// ---- 01_Equipement_Library/Sensors/TOR/FB_TOR_Spd.TcPOU
FUNCTION_BLOCK FB_TOR_Spd EXTENDS FB_TOR_Base
//////////////////
//  Surge Protection Device
//////////////////
VAR_INPUT PERSISTENT
	// Parameters of the Object (instance/model specific) 
	ParamTempoEs :TIME:=T#5S;(*  (s)Tempo before raising an alarm*)
END_VAR

VAR_OUTPUT
	//Child objects
	
END_VAR

VAR_INPUT
	// I/O Inputs 		                                     				
		
			MesDataExd			: TOR_Standard ;  

END_VAR

VAR
	//M_ALARMMANAGEMENT VARIABLES//
		FB_PermAlarm				: SR ;					// (NA) FB to maintain Fire Alarm even if sensor stop detection (burn) .
		TON_ES						: TON ; 
 
	//M_STATEMANAGER VARIABLES//

		
END_VAR

METHOD M_AlarmManagement
//////////////////
// Manages Smoke detector alarms and warnings
/////////////////

VAR 
	// Method local variables (reinitialized at each cycle) 
	FB_AlarmCodeManager			: FB_AlarmCodeManager ; 

END_VAR
// Detection Variables
TON_ES(IN:= MesDataExd.MesData.MesAlarmState , PT:= ParamTempoEs ) ; 
FB_PermAlarm(SET1 := TON_ES.Q  , Reset := CmdClearFault_G OR IN_CmdReset_L ); // SR FB for keep fire if burn .

// ALARM CODE //
	FB_AlarmCodeManager(
		bAlarm1			:= FB_PermAlarm.Q1 ,  														// Surge protection triggered	
		bAlarm2			:= SEL(ParamNbSensors<>1,FALSE, IN_MesState1_IO <> IN_MesState2_IO), 		// UNcoherent measure
		bAlarm3			:=FALSE, 																	// 
		bAlarm4			:=FALSE, 																	// 
		bAlarm5			:=FALSE, 																	//	
		bAlarm6			:=FALSE,                                                                    //
		bAlarm7			:=FALSE,                                                                    //
		bAlarm8			:=FALSE,                                                                    //
		bAlarm9			:=FALSE,                                                                    //
		bAlarm10		:=FALSE,                                                                    //
		bAlarm11		:=FALSE,                                                                    //
		bAlarm12		:=FALSE,                                                                    //
		bAlarm13		:=FALSE,                                                                    //
		bAlarm14		:=FALSE,                                                                    //
		bAlarm15		:=FALSE,                                                                    //
		wAlarmCode		=>MesDataExd.MesData.MesAlarmCode );
		
// WARNING CODE //
	FB_AlarmCodeManager(
		bAlarm1			:= IN_MesState1_IO OR  IN_MesState2_IO,	  									// At least one detector is ON 
		bAlarm2			:=FALSE, 																	// 
		bAlarm3			:=FALSE, 																	// 
		bAlarm4			:=FALSE, 																	// 
		bAlarm5			:=FALSE, 																	//
		bAlarm6			:=FALSE,        															//
		bAlarm7			:=FALSE,        															//
		bAlarm8			:=FALSE,        															//
		bAlarm9			:=FALSE,        															//
		bAlarm10		:=FALSE,        															//
		bAlarm11		:=FALSE,        															//
		bAlarm12		:=FALSE,        															//
		bAlarm13		:=FALSE,        															//
		bAlarm14		:=FALSE,        															//
		bAlarm15		:=FALSE,        															//
		wAlarmCode			=>MesDataExd.MesData.MesWarningCode);
		
// EVENT CODE //
	FB_AlarmCodeManager(
		bAlarm1			:= IN_MesState1_IO, 															// First sensor is ON
		bAlarm2			:= IN_MesState2_IO, 															// Second sensor is ON
		bAlarm3			:= FALSE, 																		// 
		bAlarm4			:= FALSE, 																		// 
		bAlarm5			:= FALSE, 																		//			
		bAlarm6			:= FALSE,                           											//
		bAlarm7			:= FALSE,                           											//
		bAlarm8			:= FALSE,                           											//
		bAlarm9			:= FALSE,                           											//
		bAlarm10		:= FALSE,                           											//
		bAlarm11		:= FALSE,                           											//
		bAlarm12		:= FALSE,                           											//
		bAlarm13		:= FALSE,                           											//
		bAlarm14		:= FALSE,                           											//
		bAlarm15		:= FALSE,                           											//
		wAlarmCode		=>MesDataExd.MesData.MesEventCode);
END_METHOD

METHOD M_Execute
//////////////////
//  Method Calls 
/////////////////

VAR 
	// Method local variables (reinitialized at each cycle) 

END_VAR

	
	IF ParamNbSensors = 9 THEN // Use of contactor bi-stable No and NC
		IN_MesState2_IO := NOT IN_MesState2_IO;
	END_IF
SUPER^.M_Execute() ;
END_METHOD

METHOD M_Init
VAR_INPUT
END_VAR
//A1_SPD_Aux.ParamAtleastOne := TRUE ; 
//A1_SPD_Aux.ParamNbSensors := 1 ; 
//A1_SPD_Aux.ParamCableCutSecurity := TRUE ;
END_METHOD

METHOD M_StateManager
//////////////////
// Detect when fire occurs
/////////////////

VAR 
	// Method local variables (reinitialized at each cycle)
 	MesStateInterm1 : BOOL;
	MesStateInterm2 : BOOL;
END_VAR

IF ParamCableCutSecurity THEN
	MesStateInterm1 := NOT IN_MesState1_IO ; 
	MesStateInterm2 := NOT IN_MesState2_IO ; 
ELSE 
	MesStateInterm1 := IN_MesState1_IO;
	MesStateInterm2 := IN_MesState2_IO;
END_IF

IF ParamNbSensors = 1 THEN 
	MesStateInterm2 := MesStateInterm1 ;
END_IF

IF ParamAtleastOne THEN 
MesDataExd.MesData.MesAlarmState := MesStateInterm1 OR MesStateInterm2 ; 
ELSE
MesDataExd.MesData.MesAlarmState := MesStateInterm1 AND MesStateInterm2 ; 
END_IF

R_TRIGAlarm(CLK:= MesDataExd.MesData.MesAlarmState ) ; 
IF R_TRIGAlarm.Q THEN
	MesCountAlarm :=  MIN(MesCountAlarm + 1 ,4294967295 ) ; 
ELSIF IN_ResetCounter THEN 
	MesCountAlarm := 0 ; 
END_IF

MesDataExd.MesData.MesCountAlarm	:= MesCountAlarm ;
END_METHOD

END_FUNCTION_BLOCK

// ---- 01_Equipement_Library/Sensors/TOR/FB_TOR_VP.TcPOU
FUNCTION_BLOCK FB_TOR_VP EXTENDS FB_TOR_Base
//////////////////
//  Voltage Presence
//////////////////

VAR_INPUT PERSISTENT
	// Parameters of the Object (instance/model specific) 
		
		
END_VAR

VAR_OUTPUT
	//Child objects
	
END_VAR

VAR_INPUT
	// I/O Inputs 		                                     				
		MesDataExd			: TOR_Standard ;  

END_VAR

VAR
	//M_ALARMMANAGEMENT VARIABLES//
		

	
END_VAR

METHOD M_AlarmManagement
//////////////////
// Manages Door sensor alarms and warnings
/////////////////

VAR 
	// Method local variables (reinitialized at each cycle) 
	FB_AlarmCodeManager : FB_AlarmCodeManager ; 


END_VAR

// ALARM CODE //
	FB_AlarmCodeManager(
 		bAlarm1			:= FALSE,    					// 
		bAlarm2			:= FALSE, 						// 
		bAlarm3			:= FALSE, 						// 
		bAlarm4			:= FALSE, 						// 
		bAlarm5			:= FALSE,       				//
		bAlarm6			:= FALSE,       				//
		bAlarm7			:= FALSE,       				//
		bAlarm8			:= FALSE,       				//
		bAlarm9			:= FALSE,       				//
		bAlarm10		:= FALSE,       				//
		bAlarm11		:= FALSE,       				//
		bAlarm12		:= FALSE,         				//
		bAlarm13		:= FALSE,         				//
		bAlarm14		:= FALSE,         				//
		bAlarm15		:= FALSE,         				//
		wAlarmCode		=>MesDataExd.MesData.MesAlarmCode);

// WARNING CODE //
	FB_AlarmCodeManager(
		bAlarm1			:= FALSE,    			// 
		bAlarm2			:= FALSE, 				//  
		bAlarm3			:= FALSE, 				//  
		bAlarm4			:= FALSE, 				//  
		bAlarm5			:= FALSE,               //
		bAlarm6			:= FALSE,               //
		bAlarm7			:= FALSE,               //
		bAlarm8			:= FALSE,               //
		bAlarm9			:= FALSE,               //
		bAlarm10		:= FALSE,               //
		bAlarm11		:= FALSE,               //
		bAlarm12		:= FALSE,               //
		bAlarm13		:= FALSE,               //
		bAlarm14		:= FALSE,               //
		bAlarm15		:= FALSE,               //
		wAlarmCode		=>MesDataExd.MesData.MesWarningCode);

// EVENT CODE //
	FB_AlarmCodeManager(
		bAlarm1			:= MesDataExd.MesData.MesAlarmState, 			//  Voltage not present anymore
		bAlarm2			:= FALSE, 							// 
		bAlarm3			:= FALSE, 							//  
		bAlarm4			:= FALSE, 							// 
		bAlarm5			:= FALSE,                           //
		bAlarm6			:= FALSE,                           //
		bAlarm7			:= FALSE,                           //
		bAlarm8			:= FALSE,                           //
		bAlarm9			:= FALSE,                           //
		bAlarm10		:= FALSE,                           //
		bAlarm11		:= FALSE,                           //
		bAlarm12		:= FALSE,                           //
		bAlarm13		:= FALSE,                           //
		bAlarm14		:= FALSE,                           //
		bAlarm15		:= FALSE,                           //
		wAlarmCode		=>MesDataExd.MesData.MesEventCode);
END_METHOD

METHOD M_StateManager
//////////////////
// Detect when fire occurs
/////////////////

VAR 
	// Method local variables (reinitialized at each cycle)
 	MesStateInterm1 : BOOL;
	MesStateInterm2 : BOOL;
END_VAR

IF ParamCableCutSecurity THEN
	MesStateInterm1 := NOT IN_MesState1_IO ; 
	MesStateInterm2 := NOT IN_MesState2_IO ; 
ELSE 
	MesStateInterm1 := IN_MesState1_IO;
	MesStateInterm2 := IN_MesState2_IO;
END_IF

IF ParamNbSensors = 1 THEN 
	MesStateInterm2 := MesStateInterm1 ;
END_IF

IF ParamAtleastOne THEN 
MesDataExd.MesData.MesAlarmState := MesStateInterm1 OR MesStateInterm2 ; 
ELSE
MesDataExd.MesData.MesAlarmState := MesStateInterm1 AND MesStateInterm2 ; 
END_IF

R_TRIGAlarm(CLK:= MesDataExd.MesData.MesAlarmState ) ; 
IF R_TRIGAlarm.Q THEN
	MesCountAlarm :=  MIN(MesCountAlarm + 1 ,4294967295 ) ; 
ELSIF IN_ResetCounter THEN 
	MesCountAlarm := 0 ; 
END_IF

MesDataExd.MesData.MesCountAlarm	:= MesCountAlarm ;
END_METHOD

END_FUNCTION_BLOCK

// ---- 01_Equipement_Library/Sensors/TOR/FB_TOR_DS.TcPOU
FUNCTION_BLOCK FB_TOR_DS EXTENDS FB_TOR_Base
//////////////////
//  Door sensor system . State = True >> Door Closed .
//////////////////

VAR_INPUT PERSISTENT
	// Parameters of the Object (instance/model specific) 
		ParamTempoDoorAlarm			: TIME := T#10S ;	(* (s) Tempo for Door sensor alarm *)
		
END_VAR

VAR_OUTPUT
	//Child objects
	
END_VAR

VAR_INPUT
	// I/O Inputs 		                                     				
	MesDataExd			: TOR_Standard ;  
		
END_VAR

VAR
	//M_ALARMMANAGEMENT VARIABLES//
		TON_Ouverture				: TON;				//(NA) Tempo to detect door opened for too long time . 



END_VAR

METHOD M_AlarmManagement
//////////////////
// Manages Door sensor alarms and warnings
/////////////////

VAR 
	// Method local variables (reinitialized at each cycle) 
	FB_AlarmCodeManager : FB_AlarmCodeManager ; 


END_VAR
// Detection Variables
TON_Ouverture(IN:= MesDataExd.MesData.MesAlarmState,PT:=ParamTempoDoorAlarm);

// ALARM CODE //
	FB_AlarmCodeManager(
 		bAlarm1			:= FALSE,    	// 
		bAlarm2			:= FALSE, 		// 
		bAlarm3			:= FALSE, 		// 
		bAlarm4			:= FALSE, 		// 
		bAlarm5			:= FALSE,       //
		bAlarm6			:= FALSE,       //
		bAlarm7			:= FALSE,       //
		bAlarm8			:= FALSE,       //
		bAlarm9			:= FALSE,       //
		bAlarm10		:= FALSE,       //
		bAlarm11		:= FALSE,       //
		bAlarm12		:= FALSE,       //
		bAlarm13		:= FALSE,       //
		bAlarm14		:= FALSE,       //
		bAlarm15		:= FALSE,       //
		wAlarmCode		=>MesDataExd.MesData.MesAlarmCode);

// WARNING CODE //
	FB_AlarmCodeManager(
		bAlarm1			:= TON_Ouverture.Q,    	// The door is opened for more than 15 seconds
		bAlarm2			:= FALSE, 				// 
		bAlarm3			:= FALSE, 				// 
		bAlarm4			:= FALSE, 				// 
		bAlarm5			:= FALSE, 				//
		bAlarm6			:= FALSE,               //
		bAlarm7			:= FALSE,               //
		bAlarm8			:= FALSE,               //
		bAlarm9			:= FALSE,               //
		bAlarm10		:= FALSE,               //
		bAlarm11		:= FALSE,               //
		bAlarm12		:= FALSE,               //
		bAlarm13		:= FALSE,               //
		bAlarm14		:= FALSE,               //
		bAlarm15		:= FALSE,               //
		wAlarmCode		=>MesDataExd.MesData.MesWarningCode);

// EVENT CODE //
	FB_AlarmCodeManager(
		bAlarm1			:= MesDataExd.MesData.MesAlarmState, 		// Door is Opened
		bAlarm2			:= FALSE, 						// 
		bAlarm3			:= FALSE, 						// 
		bAlarm4			:= FALSE, 						// 
		bAlarm5			:= FALSE, 						//
		bAlarm6			:= FALSE, 						//
		bAlarm7			:= FALSE, 						//
		bAlarm8			:= FALSE, 						//
		bAlarm9			:= FALSE, 						//
		bAlarm10		:= FALSE, 						//
		bAlarm11		:= FALSE, 						//
		bAlarm12		:= FALSE, 						//
		bAlarm13		:= FALSE, 						//
		bAlarm14		:= FALSE, 						//
		bAlarm15		:= FALSE, 						//
		wAlarmCode		=>MesDataExd.MesData.MesEventCode);
END_METHOD

METHOD M_Execute
//////////////////
//  Method Calls 
/////////////////

VAR 
	// Method local variables (reinitialized at each cycle) 
	
END_VAR


SUPER^.M_Execute() ;
END_METHOD

METHOD M_StateManager
//////////////////
// Detect when fire occurs
/////////////////

VAR 
	// Method local variables (reinitialized at each cycle)
 	MesStateInterm1 : BOOL;
	MesStateInterm2 : BOOL;
END_VAR

IF ParamCableCutSecurity THEN
	MesStateInterm1 := NOT IN_MesState1_IO ; 
	MesStateInterm2 := NOT IN_MesState2_IO ; 
ELSE 
	MesStateInterm1 := IN_MesState1_IO;
	MesStateInterm2 := IN_MesState2_IO;
END_IF

IF ParamNbSensors = 1 THEN 
	MesStateInterm2 := MesStateInterm1 ;
END_IF

IF ParamAtleastOne THEN 
MesDataExd.MesData.MesAlarmState := MesStateInterm1 OR MesStateInterm2 ; 
ELSE
MesDataExd.MesData.MesAlarmState := MesStateInterm1 AND MesStateInterm2 ; 
END_IF

R_TRIGAlarm(CLK:= MesDataExd.MesData.MesAlarmState ) ; 
IF R_TRIGAlarm.Q THEN
	MesCountAlarm :=  MIN(MesCountAlarm + 1 ,4294967295 ) ; 
ELSIF IN_ResetCounter THEN 
	MesCountAlarm := 0 ; 
END_IF

MesDataExd.MesData.MesCountAlarm	:= MesCountAlarm ;
END_METHOD

END_FUNCTION_BLOCK

// ---- 01_Equipement_Library/Sensors/TOR/FB_TOR_Rain.TcPOU
FUNCTION_BLOCK FB_TOR_Rain EXTENDS FB_TOR_Base
//////////////////
//  Rain sensor system.
//////////////////

VAR_INPUT PERSISTENT
	// Parameters of the Object (instance/model specific) 
	ParamRainPerPulse				: REAL := 10 ; (* (mm) Number of mm of rain per pulse		*)
END_VAR

VAR_OUTPUT
	//Child objects
	
END_VAR

VAR_INPUT
	// I/O Inputs 		                                     				
    ParamVarHrWarning   			: REAL :=8 ;  // (mm) Max of raining before warning mm of rain for last hour --> Mean it is raining a lot  Defaut value 8       
    ParamVarDayWarning  			: REAL :=48;  // (mm )max of raining before warning mm of rain for last day  --> Mean it rained a lot during 1 day defaut value 48
	ParamVarMinAlarm				: REAL :=-5;  // (%)  Config : Minimal allowed Site Hygrometry 



	MesDataExd			: TOR_Rain;
END_VAR

VAR


	//M_ALARMMANAGEMENT VARIABLES//
		WarningDay					: BOOL;
		WarningHr					: BOOL;
		WarningValue				: BOOL;
	
	
	//M_Execute
		FB_AverageHr				: FB_Average; 	
	    FB_AverageDay               : FB_Average;
	    FB_AverageMonth             : FB_Average;
		CTUHr						: CTU;
		CTUDay						: CTU;
		CTUMonth					: CTU;
		Hour 						: INT;
		PluvioHr_Avg		        : REAL ; 
		PluvioDay_Avg		        : REAL ; 
		PluvioMonth_Avg		        : REAL ;     
		PluvioHr_Max		        : REAL;
		PluvioDay_Max		        : REAL ; 
		PluvioMonth_Max		        : REAL ; 
        PluvioHr					: REAL ; 
		PluvioDay					: REAL ; 
		PluvioMonth					: REAL ; 

	
	
END_VAR

METHOD M_AlarmManagement
//////////////////
// Manages Door sensor alarms and warnings
/////////////////

VAR 
	// Method local variables (reinitialized at each cycle) 
	FB_AlarmCodeManager : FB_AlarmCodeManager ; 
END_VAR
	WarningDay	:= PluvioDay >= ParamVarDayWarning;
	WarningHr	:= PluvioHr >= ParamVarHrWarning;
	WarningValue:= PluvioDay <= ParamVarMinAlarm OR PluvioHr <= ParamVarMinAlarm;

// ALARM CODE //
	FB_AlarmCodeManager(
 		bAlarm1			:= FALSE,    								// 
		bAlarm2			:= FALSE, 									// 
		bAlarm3			:= FALSE, 									// 
		bAlarm4			:= FALSE, 									// 
		bAlarm5			:= FALSE,     								//
		bAlarm6			:= FALSE,  									//
		bAlarm7			:= FALSE,  									//
		bAlarm8			:= FALSE,  									//
		bAlarm9			:= FALSE,    								// 
		bAlarm10		:= FALSE, 									// 
		bAlarm11		:= FALSE, 									// 
		bAlarm12		:= FALSE, 									// 
		bAlarm13		:= FALSE,									// 
		bAlarm14		:= FALSE,									// 
		bAlarm15		:= FALSE,									// 
		wAlarmCode		=>MesDataExd.MesData.MesAlarmCode);

// WARNING CODE //
	FB_AlarmCodeManager(
		bAlarm1			:= WarningHr,   							// Raining too hard 
		bAlarm2			:= WarningDay, 								// Raining a lot during one day
		bAlarm3			:= WarningValue, 							// Raining value not coherent
		bAlarm4			:= FALSE, 									// 
		bAlarm5			:= FALSE,    								// 
		bAlarm6			:= FALSE, 									// 
		bAlarm7			:= FALSE, 									// 
		bAlarm8			:= FALSE, 									// 
		bAlarm9			:= FALSE,    								// 
		bAlarm10		:= FALSE, 									// 
		bAlarm11		:= FALSE, 									// 
		bAlarm12		:= FALSE, 									// 
		bAlarm13		:= FALSE,									// 
		bAlarm14		:= FALSE,									// 
		bAlarm15		:= FALSE,									// 
		wAlarmCode		=>MesDataExd.MesData.MesWarningCode);

// EVENT CODE //
	FB_AlarmCodeManager(
		bAlarm1			:= MesDataExd.MesData.MesAlarmState, 		// 0.2mm of water falled
		bAlarm2			:= FALSE, 									// 
		bAlarm3			:= FALSE, 									// 
		bAlarm4			:= FALSE, 									// 
		bAlarm5			:= FALSE, 									// 
		bAlarm6			:= FALSE, 									// 
		bAlarm7			:= FALSE, 									// 
		bAlarm8			:= FALSE, 									// 
		bAlarm9			:= FALSE, 									// 
		bAlarm10		:= FALSE, 									// 
		bAlarm11		:= FALSE, 									// 
		bAlarm12		:= FALSE, 									// 
		bAlarm13		:= FALSE, 									// 
		bAlarm14		:= FALSE, 									//  
		bAlarm15		:= FALSE, 									//  
		wAlarmCode		=>MesDataExd.MesData.MesEventCode);
END_METHOD

METHOD M_Execute
//////////////////
//  Method Calls 
/////////////////

VAR 
	// Method local variables (reinitialized at each cycle) 
	
END_VAR
// EMULATOR I/O //

//MAIN CODE HERE
Hour 							:=CstCycleTime_G/1000/3600  ;                        

CTUHr   (CU:= MesDataExd.MesData.MesAlarmState , RESET :=  Hour MOD 1 = 0) ; 
CTUDay  (CU:= MesDataExd.MesData.MesAlarmState , RESET := Hour MOD 24 = 0 ) ; 
CTUMonth(CU:= MesDataExd.MesData.MesAlarmState , RESET := Hour MOD 24*30 = 0 ) ; 

PluvioHr_Max := SEL( Hour MOD 1 = 0  ,   PluvioHr_Max , PluvioHr_Max:= PluvioHr)  ; 
PluvioHr := CTUHr.CV * ParamRainPerPulse ; 

PluvioDay_Max := SEL( Hour MOD 24 = 0  ,   PluvioDay_Max , PluvioDay_Max:= PluvioDay)  ; 
PluvioDay := CTUDay.CV * ParamRainPerPulse ; 

PluvioMonth_Max := SEL( Hour MOD 24*30 = 0  ,   PluvioMonth_Max , PluvioMonth_Max:= PluvioMonth)  ; 
PluvioMonth := CTUMonth.CV * ParamRainPerPulse ; 


//FB_AverageHr(ValueIn:=PluvioHr_Max  , WindowDuration := 24*3600*1000 , ValueOut => PluvioHr_Avg) ; 
//FB_AverageDay(ValueIn:=PluvioDay_Max  , WindowDuration := 24*30*3600*1000 , ValueOut => PluvioDay_Avg) ; 
//FB_AverageMonth(ValueIn:=PluvioMonth_Max  , WindowDuration := 24*365*3600*1000 , ValueOut => PluvioMonth_Avg) ;
//EVALUATE

MesDataExd.MesRainFall_LastHour 	:= PluvioHr;
MesDataExd.MesRainFall_LastDay		:= PluvioDay;
MesDataExd.MesRainFall_LastMonth	:= PluvioMonth;
MesDataExd.AvgmmHour				:= PluvioHr_Avg;
MesDataExd.AvgmmDay					:= PluvioDay_Avg;
MesDataExd.AvgmmMonth				:= PluvioMonth_Avg;

SUPER^.M_Execute();
END_METHOD

METHOD M_StateManager
//////////////////
// Detect when fire occurs
/////////////////

VAR 
	// Method local variables (reinitialized at each cycle)
 	MesStateInterm1 : BOOL;
	MesStateInterm2 : BOOL;
END_VAR

IF ParamCableCutSecurity THEN
	MesStateInterm1 := NOT IN_MesState1_IO ; 
	MesStateInterm2 := NOT IN_MesState2_IO ; 
ELSE 
	MesStateInterm1 := IN_MesState1_IO;
	MesStateInterm2 := IN_MesState2_IO;
END_IF

IF ParamNbSensors = 1 THEN 
	MesStateInterm2 := MesStateInterm1 ;
END_IF

IF ParamAtleastOne THEN 
MesDataExd.MesData.MesAlarmState := MesStateInterm1 OR MesStateInterm2 ; 
ELSE
MesDataExd.MesData.MesAlarmState := MesStateInterm1 AND MesStateInterm2 ; 
END_IF

R_TRIGAlarm(CLK:= MesDataExd.MesData.MesAlarmState ) ; 
IF R_TRIGAlarm.Q THEN
	MesCountAlarm :=  MIN(MesCountAlarm + 1 ,4294967295 ) ; 
ELSIF IN_ResetCounter THEN 
	MesCountAlarm := 0 ; 
END_IF

MesDataExd.MesData.MesCountAlarm	:= MesCountAlarm ;
END_METHOD

END_FUNCTION_BLOCK

// ---- 01_Equipement_Library/Sensors/TOR/FB_TOR_SD.TcPOU
FUNCTION_BLOCK FB_TOR_SD EXTENDS FB_TOR_Base
//////////////////
//  Smoke and Fire detection system with Typhoon triggering system. 
//////////////////
VAR_INPUT PERSISTENT
	// Parameters of the Object (instance/model specific) 
	ParamTempoFire :TIME:=T#2S;(*  (s)Tempo before raising an alarm*)
END_VAR

VAR_OUTPUT
	//Child objects
		OUT_FireDetection	: BOOL;
END_VAR

VAR_INPUT
	// I/O Inputs 		                                     				
		
		MesDataExd			: TOR_Standard ;  

END_VAR

VAR
	//M_ALARMMANAGEMENT VARIABLES//
		FB_PermAlarm				: SR ;					// (NA) FB to maintain Fire Alarm even if sensor stop detection (burn) .
		TON_Fire					: TON ; 
 
	//M_STATEMANAGER VARIABLES//
		
END_VAR

METHOD M_AlarmManagement
//////////////////
// Manages Smoke detector alarms and warnings
/////////////////

VAR 
	// Method local variables (reinitialized at each cycle) 
	FB_AlarmCodeManager			: FB_AlarmCodeManager ; 
	bTrigDaily 					: BOOL;
END_VAR
// Detection Variables
TON_Fire(IN:= MesDataExd.MesData.MesAlarmState, PT:= ParamTempoFire ) ; 
FB_PermAlarm(SET1 := TON_Fire.Q  , Reset := CmdClearFault_G OR IN_CmdReset_L ); // SR FB for keep fire if burn .

bTrigDaily := (CalLocalTimeStruct.wHour = 10 OR CalLocalTimeStruct.wHour = 16) AND CalLocalTimeStruct.wMinute = 0;

OUT_FireDetection 	:= FB_PermAlarm.Q1;

IF IN_CmdReset_L THEN
	IN_CmdReset_L := FALSE;
END_IF

// ALARM CODE //
	FB_AlarmCodeManager(
		bAlarm1			:= OUT_FireDetection ,  				// Fire Detection		
		bAlarm2			:= bTrigDaily AND OUT_FireDetection,	// Reminder : fire detection still active. 
		bAlarm3			:=FALSE, 								// 
		bAlarm4			:=FALSE, 								// 
		bAlarm5			:=FALSE, 								//
		bAlarm6			:=FALSE,                            	//
		bAlarm7			:=FALSE,                            	//
		bAlarm8			:=FALSE,                            	//
		bAlarm9			:=FALSE,                            	//
		bAlarm10		:=FALSE,                            	//
		bAlarm11		:=FALSE,                            	//
		bAlarm12		:=FALSE,                            	//
		bAlarm13		:=FALSE,                            	//
		bAlarm14		:=FALSE,                            	//
		bAlarm15		:=FALSE,                            	//
		wAlarmCode		=>MesDataExd.MesData.MesAlarmCode );
		
// WARNING CODE //
	FB_AlarmCodeManager(
		bAlarm1			:=FALSE,	  															// 
		bAlarm2			:=FALSE, 																//
		bAlarm3			:=FALSE, 																// 
		bAlarm4			:=FALSE, 																// 
		bAlarm5			:=FALSE, 																// 
		bAlarm6			:=FALSE,                                                                //
		bAlarm7			:=FALSE,                                                                //
		bAlarm8			:=FALSE,                                                                //
		bAlarm9			:=FALSE,                                                                //
		bAlarm10		:=FALSE,                                                                //
		bAlarm11		:=FALSE,                                                                //
		bAlarm12		:=FALSE,                                                                //
		bAlarm13		:=FALSE,                                                                //
		bAlarm14		:=FALSE,                                                                //
		bAlarm15		:=FALSE,                                                                //
		wAlarmCode			=>MesDataExd.MesData.MesWarningCode);
		
// EVENT CODE //
	FB_AlarmCodeManager(
		bAlarm1			:= IN_MesState1_IO, 		// First sensor is ON
		bAlarm2			:= IN_MesState2_IO, 		// Second sensor is ON
		bAlarm3			:= FALSE, 					// 		
		bAlarm4			:= FALSE, 					// 
		bAlarm5			:= FALSE, 					//
		bAlarm6			:= FALSE,                   //
		bAlarm7			:= FALSE,                   //
		bAlarm8			:= FALSE,                   //
		bAlarm9			:= FALSE,                   //
		bAlarm10		:= FALSE,                   //
		bAlarm11		:= FALSE,                   //
		bAlarm12		:= FALSE,                   //
		bAlarm13		:= FALSE,                   //
		bAlarm14		:= FALSE,                   //
		bAlarm15		:= FALSE,                   //
		wAlarmCode		=>MesDataExd.MesData.MesEventCode);
END_METHOD

METHOD M_Execute
//////////////////
//  Method Calls 
/////////////////

VAR 
	// Method local variables (reinitialized at each cycle) 

END_VAR

	IF ParamNbSensors = 9 THEN // Use of contactor bi-stable No and NC
		IN_MesState2_IO := NOT IN_MesState2_IO;
	END_IF
SUPER^.M_Execute() ;
END_METHOD

METHOD M_StateManager
//////////////////
// Detect when fire occurs
/////////////////

VAR 
	// Method local variables (reinitialized at each cycle)
 	MesStateInterm1 : BOOL;
	MesStateInterm2 : BOOL;
END_VAR

IF ParamCableCutSecurity THEN
	MesStateInterm1 := NOT IN_MesState1_IO ; 
	MesStateInterm2 := NOT IN_MesState2_IO ; 
ELSE 
	MesStateInterm1 := IN_MesState1_IO;
	MesStateInterm2 := IN_MesState2_IO;
END_IF

IF ParamNbSensors = 1 THEN 
	MesStateInterm2 := MesStateInterm1 ;
END_IF

IF ParamAtleastOne THEN 
MesDataExd.MesData.MesAlarmState := MesStateInterm1 OR MesStateInterm2 ; 
ELSE
MesDataExd.MesData.MesAlarmState := MesStateInterm1 AND MesStateInterm2 ; 
END_IF

R_TRIGAlarm(CLK:= MesDataExd.MesData.MesAlarmState ) ; 
IF R_TRIGAlarm.Q THEN
	MesCountAlarm :=  MIN(MesCountAlarm + 1 ,4294967295 ) ; 
ELSIF IN_ResetCounter THEN 
	MesCountAlarm := 0 ; 
END_IF

MesDataExd.MesData.MesCountAlarm	:= MesCountAlarm ;
END_METHOD

END_FUNCTION_BLOCK

// ---- 01_Equipement_Library/Sensors/TOR/FB_TOR_ToS.TcPOU
FUNCTION_BLOCK FB_TOR_ToS EXTENDS FB_TOR_Base
//////////////////
//  Technician on site selectOR   
//////////////////

VAR_INPUT PERSISTENT
	// Parameters of the Object (instance/model specific) 
	ParamTempoToSAlarm				: TIME := T#180M ; 	(*(min) Tempo (2h30) after ToS without clear fault >> alarm *)
	ParamTempoToSWarning			: TIME := T#120M ;  (* (min) Tempo (2h) after ToS without clear fault  >> warning*)
END_VAR

VAR_OUTPUT
	//Child objects
	
END_VAR

VAR_INPUT
	// I/O Inputs 		                                     				
	MesDataExd			: TOR_Standard ;                              			
	          	

END_VAR

VAR
	//M_ALARMMANAGEMENT VARIABLES//
		TON 						: TON ;  			 // (NA) Calculate time since technician presence activation. 
		        

	

		
END_VAR

METHOD M_AlarmManagement
//////////////////
// Manages Smoke detector alarms and warnings
/////////////////

VAR 
	// Method local variables (reinitialized at each cycle) 
	FB_AlarmCodeManager : FB_AlarmCodeManager ; 
	
END_VAR
// Detection Variables
	TON(IN:= MesDataExd.MesData.MesAlarmState AND NOT CmdClearFault_G , PT:=ParamTempoToSAlarm);   			// Reset tempo if reset commAND  
	
// ALARM CODE //
	FB_AlarmCodeManager(
		bAlarm1			:= TON.Q ,													// If technician presence is active for more than 6 hours . 				
		bAlarm2			:=FALSE, 													// 
		bAlarm3			:=FALSE, 													// 
		bAlarm4			:=FALSE, 													// 
		bAlarm5			:=FALSE, 													//
		bAlarm6			:=FALSE,        											//
		bAlarm7			:=FALSE,        											//
		bAlarm8			:=FALSE,        											//
		bAlarm9			:=FALSE,        											//
		bAlarm10		:=FALSE,        											//
		bAlarm11		:=FALSE,        											//
		bAlarm12		:=FALSE,        											//
		bAlarm13		:=FALSE,        											//
		bAlarm14		:=FALSE,        											//
		bAlarm15		:=FALSE,        											//
		wAlarmCode		=>MesDataExd.MesData.MesAlarmCode);

// WARNING CODE //
	FB_AlarmCodeManager(
		bAlarm1			:= TON.ET > ParamTempoToSWarning ,				// If technician presence is active for more than 2 hours .  
		bAlarm2			:=FALSE, 										// 
		bAlarm3			:=FALSE, 										// 
		bAlarm4			:=FALSE, 										// 
		bAlarm5			:=FALSE, 										//
		bAlarm6			:=FALSE,        								//
		bAlarm7			:=FALSE,        								//
		bAlarm8			:=FALSE,        								//
		bAlarm9			:=FALSE,        								//
		bAlarm10		:=FALSE,        								//
		bAlarm11		:=FALSE,        								//
		bAlarm12		:=FALSE,        								//
		bAlarm13		:=FALSE,        								//
		bAlarm14		:=FALSE,        								//
		bAlarm15		:=FALSE,        								//
		wAlarmCode		=>MesDataExd.MesData.MesWarningCode);
			
// EVENT CODE //
	FB_AlarmCodeManager(
		bAlarm1			:= MesDataExd.MesData.MesAlarmState, 		// Technician On Site
		bAlarm2			:= FALSE, 						// 
		bAlarm3			:= FALSE, 						// 
		bAlarm4			:= FALSE, 						// 
		bAlarm5			:= FALSE, 						//
		bAlarm6			:= FALSE, 						//
		bAlarm7			:= FALSE,                       //
		bAlarm8			:= FALSE,                       //
		bAlarm9			:= FALSE,                       //
		bAlarm10		:= FALSE,                       //
		bAlarm11		:= FALSE,                       //
		bAlarm12		:= FALSE,                       //
		bAlarm13		:= FALSE,                       //
		bAlarm14		:= FALSE,                       //
		bAlarm15		:= FALSE,                       //
		wAlarmCode		=>MesDataExd.MesData.MesEventCode);
END_METHOD

METHOD M_Execute
//////////////////
//  Method Calls 
/////////////////

VAR 
	// Method local variables (reinitialized at each cycle) 

END_VAR
// EMULATOR I/O //

SUPER^.M_Execute() ;
END_METHOD

METHOD M_StateManager
//////////////////
// Detect when fire occurs
/////////////////

VAR 
	// Method local variables (reinitialized at each cycle)
 	MesStateInterm1 : BOOL;
	MesStateInterm2 : BOOL;
END_VAR

IF ParamCableCutSecurity THEN
	MesStateInterm1 := NOT IN_MesState1_IO ; 
	MesStateInterm2 := NOT IN_MesState2_IO ; 
ELSE 
	MesStateInterm1 := IN_MesState1_IO;
	MesStateInterm2 := IN_MesState2_IO;
END_IF

IF ParamNbSensors = 1 THEN 
	MesStateInterm2 := MesStateInterm1 ;
END_IF

IF ParamAtleastOne THEN 
MesDataExd.MesData.MesAlarmState := MesStateInterm1 OR MesStateInterm2 ; 
ELSE
MesDataExd.MesData.MesAlarmState := MesStateInterm1 AND MesStateInterm2 ; 
END_IF

R_TRIGAlarm(CLK:= MesDataExd.MesData.MesAlarmState ) ; 
IF R_TRIGAlarm.Q THEN
	MesCountAlarm :=  MIN(MesCountAlarm + 1 ,4294967295 ) ; 
ELSIF IN_ResetCounter THEN 
	MesCountAlarm := 0 ; 
END_IF

MesDataExd.MesData.MesCountAlarm	:= MesCountAlarm ;
END_METHOD

END_FUNCTION_BLOCK

// ---- 01_Equipement_Library/TAC/FB_TAC.TcPOU
FUNCTION_BLOCK FB_TAC

VAR_INPUT PERSISTENT
		ParamTONFiltering						: TIME:=T#200MS; 	(* (ms) Minimum tempo filter before command validation (noise filtering)*)
		ParamDurationPulse						: TIME:= T#2S;		(* (ms) Duration of the output pulses *)
	MesDataExd					: TAC_Standard;	
END_VAR

VAR_INPUT
	IN_CmdOn_IO					: BOOL;		(* Order coming from Grid Manager *)
	IN_CmdOff_IO				: BOOL;		(* Order coming from Grid Manager *)
	IN_MesOn_IO					: BOOL;		(* Measure from equipment *)
	IN_MesOff_IO				: BOOL;		(* Measure from equipment *)
	IN_MesFault_IO				: BOOL;
	
	IN_CmdDisconnect_IO			: BOOL;
	
	IN_CmdOn_Other				: BOOL;
	IN_CmdOff_Other				: BOOL;
	
	IN_CmdReset					: BOOL;
	
END_VAR
VAR_OUTPUT
	OUT_CmdDisconnect_IO		: BOOL;
	OUT_CmdOn_IO				: BOOL;	
	OUT_CmdOff_IO				: BOOL;
	OUT_MesFault_IO				: BOOL;
	OUT_CmdH1_IO				: BOOL; // Envoi commande H1 au Relais de Protection
END_VAR

VAR PERSISTENT
END_VAR

VAR
	
	TONCmdOn					: TON;
	TONCmdOff					: TON;
	TONCmdOnAck					: TON;
	TONCmdOffAck				: TON;
	
	R_TRIG_MesOn				: R_TRIG;
	F_TRIG_MesOn				: F_TRIG;
	
	TP_CmdOn					: TP;
	TP_CmdOff					: TP;

	
END_VAR

METHOD M_AlarmManagement
//////////////////
// alarm and warning management
/////////////////

VAR 
	FB_AlarmCodeManager			: FB_AlarmCodeManager ; 
	
END_VAR
FB_AlarmCodeManager
(               
	bAlarm1  := MesDataExd.MesData.OUT_CmdActivated,		// TAC Activated 
	bAlarm2  := IN_MesOn_IO,					// TAC is ON : Ack from equipment
	bAlarm3  := MesDataExd.MesData.MesFault,	// Fault on TAC
	bAlarm4  := OUT_CmdH1_IO,					// Protection relay switched to H1
	bAlarm5  := IN_CmdDisconnect_IO,			// Disconnect order from TAC
	bAlarm6  := IN_MesOff_IO,					// TAC is OFF : Ack from equipment
	bAlarm7  := FALSE,
	bAlarm8  := FALSE,
	bAlarm9  := FALSE,
	bAlarm10 := FALSE,
	bAlarm11 := FALSE,
	bAlarm12 := FALSE,
	bAlarm13 := FALSE,
	bAlarm14 := FALSE,
	bAlarm15 := FALSE,
	wAlarmCode =>MesDataExd.MesData.mesAlarmCode
);

FB_AlarmCodeManager
(               
	bAlarm1  := FALSE,
	bAlarm2  := NOT MesDataExd.MesData.OUT_CmdActivated,		// TAC Deactivated 
	bAlarm3  := FALSE,
	bAlarm4  := FALSE,
	bAlarm5  := FALSE,
	bAlarm6  := FALSE,
	bAlarm7  := FALSE,
	bAlarm8  := FALSE,
	bAlarm9  := FALSE,
	bAlarm10 := FALSE,
	bAlarm11 := FALSE,
	bAlarm12 := FALSE,
	bAlarm13 := FALSE,
	bAlarm14 := FALSE,
	bAlarm15 := FALSE,
	wAlarmCode =>MesDataExd.MesData.MesWarningCode
);
END_METHOD

METHOD M_Evaluate
//////////////////
//  Evaluate grid variables 
/////////////////
VAR 
	// Method local variables (reinitialized at each cycle) 
	WatchDog	: BOOL;
END_VAR

//Filtering Input
TONCmdOn			(IN:=IN_CmdOn_IO		,PT:=ParamTONFiltering);	
TONCmdOff			(IN:=IN_CmdOff_IO		,PT:=ParamTONFiltering);	
TONCmdOnAck			(IN:=IN_MesOn_IO		,PT:=ParamTONFiltering);	
TONCmdOffAck		(IN:=IN_MesOff_IO	,PT:=ParamTONFiltering);

IF IN_CmdReset OR CmdClearFault_G THEN
	MesDataExd.MesData.MesFault := FALSE;
END_IF

//Logical Equation
	(* Command to switch TAC ON from GRID or OPC*)
		IF TONCmdOn.Q OR IN_CmdOn_Other THEN
			MesDataExd.MesData.OUT_CmdActivated := TRUE;
			OUT_CmdOn_IO := TRUE;
			OUT_CmdOff_IO := FALSE;
		END_IF
		
	(* Command to switch TAC OFF from GRID or OPC*)
		IF TONCmdOff.Q OR IN_CmdOff_Other THEN
			MesDataExd.MesData.OUT_CmdActivated := FALSE;
			OUT_CmdOn_IO := FALSE;
			OUT_CmdOff_IO := TRUE;
		END_IF
		
	(* Fault received from TAC*) 	
		IF IN_MesFault_IO THEN
			MesDataExd.MesData.MesFault := TRUE ;
		END_IF

// Send orders to TAC:
	R_TRIG_MesOn(CLK := MesDataExd.MesData.MesActivated);
	F_TRIG_MesOn(CLK := MesDataExd.MesData.MesActivated);
	
	TP_CmdOn(IN := R_TRIG_MesOn.Q, pt := ParamDurationPulse);
	TP_CmdOff(IN := F_TRIG_MesOn.Q, pt := ParamDurationPulse);
	
	OUT_CmdH1_IO := MesDataExd.MesData.OUT_CmdActivated;
END_METHOD

METHOD M_Execute : BOOL
VAR_INPUT
END_VAR

	M_Evaluate() ; 
	M_AlarmManagement();
END_METHOD

END_FUNCTION_BLOCK

// ---- 01_Equipement_Library/Tariff Meter/FB_EM_Base.TcPOU
FUNCTION_BLOCK FB_EM_Base
//////////////////
// Measurement Solution. Base FB
//////////////////
VAR_INPUT PERSISTENT
	// Parameters of the Object (instance specific) 
		CmdInitialValues			: EM_Standard;
	{attribute 'OPC.UA.DA' := '1'} 
		ParamStepEactCons			: REAL := 10;	// kWh step for tariff meter
	{attribute 'OPC.UA.DA' := '1'}                  
		ParamStepEactProd			: REAL := 10;   // kWh step for tariff meter
	{attribute 'OPC.UA.DA' := '1'}                  
		ParamStepEreactCons			: REAL := 10;   // kVArh step for tariff meter
	{attribute 'OPC.UA.DA' := '1'}                  
		ParamStepEreactProd			: REAL := 10;   // kVArh step for tariff meter
		ParamEssNum					: UINT :=1 ; 	// ESS Num
END_VAR

VAR_INPUT
	//Child objects
		IN_CmdReset_L					: BOOL;			// (NA) Local reset of the alarms	
END_VAR                                                             
VAR                                                                 
	//M_ALARMMANAGEMENT VARIABLES//                                 
		TON_ComAlarm				: TON ; 			// Tempo before deteting loss of communication. 
                                                        
	//M_INIT VARIABLES //                               
		bInit						: BOOL 	:= TRUE ; 	// (NA) Initialize object parameters at first cycle 
		                                                
	// M_EXECUTE VARIABLES //                           
 //	MesDataExd			: EM;					// (NA) Structure of the Tariff Meter
		MesCP_Read					: BOOL := TRUE;	(* Read function enable *)
		MesCP_Write					: BOOL := TRUE;	(* Write function enable *)                                                
	// M_EVALUATE VARIABLES //                          
		trig1 						: R_TRIG;			// (NA) Trigger for the pulses
		trig2 						: R_TRIG;			// (NA) Trigger for the pulses
		trig3 						: R_TRIG;			// (NA) Trigger for the pulses
		trig4 						: R_TRIG;			// (NA) Trigger for the pulses

                      
END_VAR

VAR_INPUT
		IN_MesPulseEactCons_IO			: BOOL;		// Pulse Input signal for the Active energy consumed measurement
		IN_MesPulseEactProd_IO			: BOOL;		// Pulse Input signal for the Active energy produced measurement
		IN_MesPulseEreactCons_IO		: BOOL;		// Pulse Input signal for the Reactive energy consumed measurement
		IN_MesPulseEreactProd_IO		: BOOL;		// Pulse Input signal for the Reactive energy produced measurement
END_VAR

METHOD M_AlarmManagement
//////////////////
// Digiware measurement tool alarm and warning management
/////////////////

VAR 
	
END_VAR
END_METHOD

METHOD M_Evaluate
VAR_INPUT
END_VAR

VAR

END_VAR
END_METHOD

METHOD M_Execute
//////////////////
//  Method Calls 
/////////////////
VAR 
	// Method local variables (reinitialized at each cycle) 
	// EMULATOR

	
END_VAR



// METHODS CALLS //
	IF bInit THEN
		M_Init() ; 
		bInit					:= FALSE ; 
	ELSIF CmdInit_G OR IN_CmdReset_L THEN 
		bInit:= TRUE ;
	END_IF

	M_Evaluate();	

	////////////////////
	M_AlarmManagement();
END_METHOD

METHOD M_Init
VAR 

END_VAR
END_METHOD

END_FUNCTION_BLOCK

// ---- 01_Equipement_Library/Tariff Meter/FB_EM_ION8650.TcPOU
FUNCTION_BLOCK FB_EM_ION8650 EXTENDS FB_EM_Base
//////////////////
// Measurement Solution. Base FB
//////////////////
VAR_INPUT PERSISTENT
	{attribute 'OPC.UA.DA' := '1'} 
	ParamTcpPort						: UINT	 := 502;				(* (NA) TCP port						 		*) 
	{attribute 'OPC.UA.DA' := '1'}  	                                	                                     		
	ParamIPAddress						: STRING := '10.0.0.1'; 		(* (NA) IP address of main gateway SC3 	 		*)
	ParamUnitID 						: BYTE   := 1; 					(* (NA) Modbus Unit ID					 		*)
	ParamTimeout						: TIME   := T#5S;		  		(* (s) Timeout for modbus reading 		 		*)
	ParamEmailOC						: BOOL   := FALSE;				(* (NA) Send email to OC in case of phase loss  *)
END_VAR

VAR_INPUT
	//Child objects
	MesDataExd			  				: EM_ION8650; 
	AlarmOn_Sent		 				: BOOL;
	AlarmOff_Sent						: BOOL;
END_VAR

VAR
	//M_ALARMMANAGEMENT VARIABLES//
	FB_DetectFixedValue   				: FB_DetectFixedValue; 
    Eact_null    		  				: REAL;                                   								
	Message_Email_SMC1		  			: ST_ValuesAlarms;
	Message_Email_SMC2		  			: ST_ValuesAlarms;
	TrigAlarmGrid_ON	  				: R_TRIG;
	TrigAlarmGrid_OFF	  				: F_TRIG;
	
	FB_ModbusRead	          			: ARRAY [1..6] OF FB_ModbusRead; 	// (NA) FB for Modbus Reading                          		
	MesBlock1_Temp						: ARRAY [1..2] OF WORD;       		// (NA) Temporary Block with multiple modbus reading (Caution : Double Word variables)	                            		
	MesBlock2_Temp						: ARRAY [1..10] OF WORD; 
	AX_ModbusReadAlarm					: ARRAY [1..2] OF BOOL;
	AX_ModbusReadAlarmId				: ARRAY [1..2] OF UDINT;
END_VAR

METHOD M_AlarmManagement
//////////////////
// Digiware measurement tool alarm and warning management
/////////////////

VAR 
	FB_AlarmCodeManager : FB_AlarmCodeManager; 
END_VAR

FB_DetectFixedValue(IN_Addr := ADR(MesDataExd.MesData.MesEactCons), IN_Size := SIZEOF(MesDataExd.MesData.MesEactCons), IN_Duration :=T#3H , IN_EmptyStruct := ADR(Eact_null ) ); 

// ALARM CODE //
	FB_AlarmCodeManager(
		bAlarm1			:= MesDataExd.MesData.MesEActProd > 10,																	// Production measured			
		bAlarm2			:= FB_DetectFixedValue.OUT_bStatic,																		// Loss of communication with meter 
		bAlarm3			:=FALSE,//MesDataExd.MesLossPhase, 																			// Loss of one or more TC phases 
		bAlarm4			:=FALSE, 																								// 
		bAlarm5			:=FALSE, 																								//
		bAlarm6			:=FALSE,        																						//
		bAlarm7			:=FALSE,        																						//
		bAlarm8			:=FALSE,        																						//
		bAlarm9			:=FALSE,        																						//
		bAlarm10		:=FALSE,        																						//
		bAlarm11		:=FALSE,        																						//
		bAlarm12		:=FALSE,        																						//
		bAlarm13		:=FALSE,        																						//
		bAlarm14		:=FALSE,        																						//
		bAlarm15		:=FALSE,        																						//
		wAlarmCode		=>MesDataExd.MesData.MesAlarmCode);

// WARNING CODE //
	FB_AlarmCodeManager(
		bAlarm1			:=FALSE,										//  
		bAlarm2			:=FALSE, 										// 
		bAlarm3			:=FALSE, 										// 
		bAlarm4			:=FALSE, 										// 
		bAlarm5			:=FALSE, 										//
		bAlarm6			:=FALSE,        								//
		bAlarm7			:=FALSE,        								//
		bAlarm8			:=FALSE,        								//
		bAlarm9			:=FALSE,        								//
		bAlarm10		:=FALSE,        								//
		bAlarm11		:=FALSE,        								//
		bAlarm12		:=FALSE,        								//
		bAlarm13		:=FALSE,        								//
		bAlarm14		:=FALSE,        								//
		bAlarm15		:=FALSE,        								//
		wAlarmCode		=>MesDataExd.MesData.MesWarningCode);
			
// EVENT CODE //
	FB_AlarmCodeManager(
		bAlarm1			:= IN_CmdReset_L, 				// Reset command
		bAlarm2			:= FALSE, 						// 
		bAlarm3			:= FALSE, 						// 
		bAlarm4			:= FALSE, 						// 
		bAlarm5			:= FALSE, 						//
		bAlarm6			:= FALSE, 						//
		bAlarm7			:= FALSE,                       //
		bAlarm8			:= FALSE,                       //
		bAlarm9			:= FALSE,                       //
		bAlarm10		:= FALSE,                       //
		bAlarm11		:= FALSE,                       //
		bAlarm12		:= FALSE,                       //
		bAlarm13		:= FALSE,                       //
		bAlarm14		:= FALSE,                       //
		bAlarm15		:= FALSE,                       //
		wAlarmCode		=>MesDataExd.MesData.MesEventCode);
		
		
IF ParamEmailOC THEN
	IF ParamTcpPort = 503 THEN // SMC1
		// Send email to OC in case of loss of a measurement phase
		TrigAlarmGrid_ON(CLK:= MesDataExd.MesLossPhase); 
		
		IF NOT MesDataExd.MesLossPhase THEN 
			AlarmOn_Sent := FALSE;
			//FUN_SendMail.FIFO.In.ID		:= 0;
		END_IF
		
		IF TrigAlarmGrid_ON.Q  AND NOT AlarmOn_Sent THEN //A1_SUBMV.A1_EM_Main.MesDataExd.MesLossPhase AND NOT AlarmOn_Sent THEN
			Message_Email_SMC1.TimeStamp_Act:= SYSTEMTIME_TO_STRING(CalLocalTimeStruct);
			Message_Email_SMC1.ID			:= 200;//65535;
			Message_Email_SMC1.Value		:= TRUE;
			FUN_SendMail.FIFO.In 			:= Message_Email_SMC1;
			FUN_SendMail.FIFO.A_Add();
		END_IF
		
		// Alarm disactivated
		TrigAlarmGrid_OFF(CLK:= MesDataExd.MesLossPhase); 
		
		IF MesDataExd.MesLossPhase THEN 
			AlarmOff_Sent := FALSE;
		END_IF
		
		IF TrigAlarmGrid_OFF.Q  AND NOT AlarmOff_Sent THEN //A1_SUBMV.A1_EM_Main.MesDataExd.MesLossPhase AND NOT AlarmOn_Sent THEN
			Message_Email_SMC1.TimeStamp_Act:= SYSTEMTIME_TO_STRING(CalLocalTimeStruct);
			Message_Email_SMC1.ID			:= 200;//65535;
			Message_Email_SMC1.Value		:= FALSE;
			FUN_SendMail.FIFO.In 			:= Message_Email_SMC1;
			FUN_SendMail.FIFO.A_Add();
		END_IF
	ELSIF ParamTcpPort = 504 THEN // SMC2
		// Send email to OC in case of loss of a measurement phase
		TrigAlarmGrid_ON(CLK:= MesDataExd.MesLossPhase); 
		
		IF NOT MesDataExd.MesLossPhase THEN 
			AlarmOn_Sent := FALSE;
		END_IF
		
		IF TrigAlarmGrid_ON.Q  AND NOT AlarmOn_Sent THEN 
			Message_Email_SMC2.TimeStamp_Act:= SYSTEMTIME_TO_STRING(CalLocalTimeStruct);
			Message_Email_SMC2.ID			:= 200;
			Message_Email_SMC2.Value		:= TRUE;
			FUN_SendMail.FIFO.In 			:= Message_Email_SMC2;
			FUN_SendMail.FIFO.A_Add();
		END_IF
		
		// Alarm disactivated
		TrigAlarmGrid_OFF(CLK:= MesDataExd.MesLossPhase); 
		
		IF MesDataExd.MesLossPhase THEN 
			AlarmOff_Sent := FALSE;
		END_IF
		
		IF TrigAlarmGrid_OFF.Q  AND NOT AlarmOff_Sent THEN 
			Message_Email_SMC2.TimeStamp_Act:= SYSTEMTIME_TO_STRING(CalLocalTimeStruct);
			Message_Email_SMC2.ID			:= 200;
			Message_Email_SMC2.Value		:= FALSE;
			FUN_SendMail.FIFO.In 			:= Message_Email_SMC2;
			FUN_SendMail.FIFO.A_Add();
		END_IF
	END_IF
END_IF
END_METHOD

METHOD M_Evaluate
VAR_INPUT
END_VAR

VAR
	TM_0 : EM_ION8650;	// Empty structure
	OutTrig_Eac : BOOL;
	OutTrig_Eap : BOOL;
	OutTrig_Erc : BOOL;
	OutTrig_Erp : BOOL;
	bTest : BOOL;
END_VAR
IF CmdInitialValues.MesData.MesEactCons <> TM_0.MesData.MesEactCons OR CmdInitialValues.MesData.MesEActProd <> TM_0.MesData.MesEActProd OR CmdInitialValues.MesData.MesEReactCons <> TM_0.MesData.MesEReactCons OR CmdInitialValues.MesData.MesEReactProd <> TM_0.MesData.MesEReactProd THEN
MesDataExd:= CmdInitialValues;
	CmdInitialValues := TM_0 ;
END_IF

trig1(CLK := IN_MesPulseEactCons_IO, Q => OutTrig_Eac);
trig2(CLK := IN_MesPulseEactProd_IO, Q => OutTrig_Eap);
trig3(CLK:= IN_MesPulseEreactCons_IO, Q => OutTrig_Erc);
trig4(CLK:= IN_MesPulseEreactProd_IO, Q => OutTrig_Erp);

IF OutTrig_Eac THEN
MesDataExd.MesData.MesEactCons := MesDataExd.MesData.MesEactCons + ParamStepEactCons;
END_IF 

IF OutTrig_Eap THEN
MesDataExd.MesData.MesEActProd := MesDataExd.MesData.MesEActProd + ParamStepEactProd;
END_IF 

IF OutTrig_Erc THEN
MesDataExd.MesData.MesEReactCons := MesDataExd.MesData.MesEReactCons + ParamStepEreactCons;
END_IF 

IF OutTrig_Erp THEN
MesDataExd.MesData.MesEReactProd := MesDataExd.MesData.MesEReactProd + ParamStepEreactProd;
END_IF 

SUPER^.M_Evaluate();
END_METHOD

METHOD M_Init
VAR 
	InitialValues : EM_ION8650; 
END_VAR

Message_Email_SMC1.Message 	:= '"SMC 1: Falta tensión en fases A, B o C en la subestación del Parque Solar Fotovoltaico Matrisol';
Message_Email_SMC2.Message 	:= '"SMC 2: Falta tensión en fases A, B o C en la subestación del Parque Solar Fotovoltaico Matrisol';
bInit 						:= FALSE;
END_METHOD


METHOD M_Read : BOOL
VAR_INPUT
END_VAR

VAR
	MW_UInt				: FB_MergeWordsToUint;
	MW_Real				: FB_MergeWordsToDint;
	Temp_Value			: UINT;
END_VAR

IF MesDataExd.MesData.MesCP_Read  THEN	
//// MODBUS Read	
	FB_ModbusRead[1]
		(
			nTCPPort		:= ParamTcpPort,
			ClockRead		:= MesDataExd.MesData.MesCP_Read AND ClockRead, 
			Reset			:= CmdClearFault_G OR IN_CmdReset_L,
			sIPAddr			:= ParamIPAddress,
			nUnitID			:= ParamUnitID, 
			tTimeout		:= ParamTimeout,
			nQuantity		:= 1, 
			nMBAddr			:= 218, 
			cbLength		:= SIZEOF(MesBlock1_Temp), 
			pDestAddr		:= ADR(MesBlock1_Temp), 
			ModbusReadAlarm	=> AX_ModbusReadAlarm[1], 
			ErrorId			=> AX_ModbusReadAlarmId[1]
		);
	
	// FB_ModbusRead[2]
	// 	(
	// 		nTCPPort		:= ParamTcpPort,
	// 		ClockRead		:= MesDataExd.MesData.MesCP_Read AND ClockRead, 
	// 		Reset			:= CmdClearFault_G OR IN_CmdReset_L,
	// 		sIPAddr			:= ParamIPAddress,
	// 		nUnitID			:= ParamUnitID, 
	// 		tTimeout		:= ParamTimeout,
	// 		nQuantity		:= 12, 
	// 		nMBAddr			:= 40091, 
	// 		cbLength		:= SIZEOF(MesBlock1_Temp), 
	// 		pDestAddr		:= ADR(MesBlock2_Temp), 
	// 		ModbusReadAlarm	=> AX_ModbusReadAlarm[2], 
	// 		ErrorId			=> AX_ModbusReadAlarmId[2]
	// 	);
	
	MW_UInt(WORD_STRONG:= MesBlock1_Temp[ 1], VAR_OUT := Temp_Value);
		
	IF Temp_Value = 2 THEN
		MesDataExd.MesLossPhase := TRUE;
	ELSE
		MesDataExd.MesLossPhase := FALSE;	
	END_IF 
	
	MW_Real(WORD_STRONG:= MesBlock2_Temp[ 2], WORD_WEAK:= MesBlock2_Temp[ 1], VAR_OUT := MesDataExd.MesData.MesEActProd);
	MW_Real(WORD_STRONG:= MesBlock2_Temp[ 2], WORD_WEAK:= MesBlock2_Temp[ 1], VAR_OUT := MesDataExd.MesData.MesEActCons);
	
END_IF
END_METHOD

END_FUNCTION_BLOCK

// ---- 01_Equipement_Library/Tariff Meter/FB_EM_Pulse.TcPOU
FUNCTION_BLOCK FB_EM_Pulse EXTENDS FB_EM_Base
//////////////////
// Measurement Solution. Base FB
//////////////////
VAR_INPUT PERSISTENT
	// Parameters of the Object (instance specific) 
		
	
END_VAR

VAR_OUTPUT
	//Child objects
	
END_VAR

VAR_INPUT
			MesDataExd			: EM_Standard ; 
END_VAR

VAR
	//M_ALARMMANAGEMENT VARIABLES//
		FB_DetectFixedValue   : FB_DetectFixedValue ; 
        Eact_null    		  : REAL ;                                   								
		

	//M_INIT VARIABLES //

		
	// M_EXECUTE VARIABLES //
 		
	// M_Reset_L
		
                      
END_VAR

VAR_INPUT
		
END_VAR

METHOD M_AlarmManagement
//////////////////
// Digiware measurement tool alarm and warning management
/////////////////

VAR 
	FB_AlarmCodeManager : FB_AlarmCodeManager ; 
END_VAR

FB_DetectFixedValue(IN_Addr := ADR(MesDataExd.MesData.MesEactCons) , IN_Size := SIZEOF(MesDataExd.MesData.MesEactCons) , IN_Duration :=T#3H , IN_EmptyStruct := ADR(Eact_null ) ); 

// ALARM CODE //
	FB_AlarmCodeManager(
		bAlarm1			:= MesDataExd.MesData.MesEActProd > 10 ,																			// Production measured			
		bAlarm2			:=FB_DetectFixedValue.OUT_bStatic 	,																	// Loss of communication with meter 
		bAlarm3			:=FALSE, 																								// 
		bAlarm4			:=FALSE, 																								// 
		bAlarm5			:=FALSE, 																								//
		bAlarm6			:=FALSE,        																						//
		bAlarm7			:=FALSE,        																						//
		bAlarm8			:=FALSE,        																						//
		bAlarm9			:=FALSE,        																						//
		bAlarm10		:=FALSE,        																						//
		bAlarm11		:=FALSE,        																						//
		bAlarm12		:=FALSE,        																						//
		bAlarm13		:=FALSE,        																						//
		bAlarm14		:=FALSE,        																						//
		bAlarm15		:=FALSE,        																						//
		wAlarmCode		=>MesDataExd.MesData.MesAlarmCode);

// WARNING CODE //

	FB_AlarmCodeManager(
		bAlarm1			:= FALSE ,										//  
		bAlarm2			:=FALSE, 										// 
		bAlarm3			:=FALSE, 										// 
		bAlarm4			:=FALSE, 										// 
		bAlarm5			:=FALSE, 										//
		bAlarm6			:=FALSE,        								//
		bAlarm7			:=FALSE,        								//
		bAlarm8			:=FALSE,        								//
		bAlarm9			:=FALSE,        								//
		bAlarm10		:=FALSE,        								//
		bAlarm11		:=FALSE,        								//
		bAlarm12		:=FALSE,        								//
		bAlarm13		:=FALSE,        								//
		bAlarm14		:=FALSE,        								//
		bAlarm15		:=FALSE,        								//
		wAlarmCode		=>MesDataExd.MesData.MesWarningCode);
			
// EVENT CODE //
	FB_AlarmCodeManager(
		bAlarm1			:= IN_CmdReset_L, 				// Reset command
		bAlarm2			:= FALSE, 						// 
		bAlarm3			:= FALSE, 						// 
		bAlarm4			:= FALSE, 						// 
		bAlarm5			:= FALSE, 						//
		bAlarm6			:= FALSE, 						//
		bAlarm7			:= FALSE,                       //
		bAlarm8			:= FALSE,                       //
		bAlarm9			:= FALSE,                       //
		bAlarm10		:= FALSE,                       //
		bAlarm11		:= FALSE,                       //
		bAlarm12		:= FALSE,                       //
		bAlarm13		:= FALSE,                       //
		bAlarm14		:= FALSE,                       //
		bAlarm15		:= FALSE,                       //
		wAlarmCode		=>MesDataExd.MesData.MesEventCode);
END_METHOD

METHOD M_Evaluate
VAR_INPUT
END_VAR

VAR
	TM_0 : EM_Standard;	// Empty structure
	OutTrig_Eac : BOOL;
	OutTrig_Eap : BOOL;
	OutTrig_Erc : BOOL;
	OutTrig_Erp : BOOL;
	bTest : BOOL;
END_VAR
IF CmdInitialValues.MesData.MesEactCons <> TM_0.MesData.MesEactCons OR CmdInitialValues.MesData.MesEActProd <> TM_0.MesData.MesEActProd OR CmdInitialValues.MesData.MesEReactCons <> TM_0.MesData.MesEReactCons OR CmdInitialValues.MesData.MesEReactProd <> TM_0.MesData.MesEReactProd THEN
MesDataExd:= CmdInitialValues;
	CmdInitialValues := TM_0 ;
END_IF

trig1(CLK := IN_MesPulseEactCons_IO, Q => OutTrig_Eac);
trig2(CLK := IN_MesPulseEactProd_IO, Q => OutTrig_Eap);
trig3(CLK:= IN_MesPulseEreactCons_IO, Q => OutTrig_Erc);
trig4(CLK:= IN_MesPulseEreactProd_IO, Q => OutTrig_Erp);

IF OutTrig_Eac THEN
MesDataExd.MesData.MesEactCons := MesDataExd.MesData.MesEactCons + ParamStepEactCons;
END_IF 

IF OutTrig_Eap THEN
MesDataExd.MesData.MesEActProd := MesDataExd.MesData.MesEActProd + ParamStepEactProd;
END_IF 

IF OutTrig_Erc THEN
MesDataExd.MesData.MesEReactCons := MesDataExd.MesData.MesEReactCons + ParamStepEreactCons;
END_IF 

IF OutTrig_Erp THEN
MesDataExd.MesData.MesEReactProd := MesDataExd.MesData.MesEReactProd + ParamStepEreactProd;
END_IF 

SUPER^.M_Evaluate();
END_METHOD

METHOD M_Init
VAR 
	InitialValues : EM_Standard ; 
END_VAR
MesDataExd := InitialValues ; 
bInit := FALSE ;
END_METHOD

END_FUNCTION_BLOCK

// ---- 01_Equipement_Library/Tracker/FB_NCU_Base.TcPOU
FUNCTION_BLOCK  FB_NCU_Base
//////////////////
// NCU Function 
//////////////////
VAR_INPUT PERSISTENT
	// Parameters of the Object (instance/model specific) 
	ParamIPAddress				: STRING := '192.168.1.1' ; // IP 
	ParamTcpPort				: UINT		:= 502;
	ParamTimeOut				: TIME := T#10S ; 
	ParamClockReadTime			: TIME := T#1S ; 
	
	ParamClockWriteTime			: TIME := T#1S ; 	
	
	ParamUnitID 				: BYTE:=1; 					// (NA)   SMA Modbus Unit ID.
	ParamNbTracker				: BYTE ; 					// Number of tracker behind the 
	ParamNCUNum					: INT ; 					// Numerous of TCU 
	                                                		
	ParamTempoComAlarm			: TIME 			 ; 			// (s) Config : Tempo to detect LOC Alarm	

END_VAR

VAR_INPUT 
	//Child objects
	IN_CmdReset_L							: BOOL;				// (NA) External Reset Command	
    IN_CmdToggleRead						: BOOL;
    IN_CmdToggleWrite						: BOOL;
END_VAR


VAR
	//M_ROTATE VARIABLES//
	
		
	//M_ALARMMANAGEMENT VARIABLES//
		TON_ComAlarm				: TON ; 												// Tempo before detecting loss of communication. 
	
	
		
	//M_READ VARAIBLES 
	
		
	//M_STATEMANAGER VARIABLES//
	
		
	// M_EXECUTE VARIABLES 	//      
		TP1							: TP ; 				// (NA) Tempo to define Modbus Reading Frequency 
		TP2 						: TP ; 				// (NA) Tempo to define Modbus Writing Frequency
		                            
		ClockRead					: BOOL;				// (NA) Modbus reading Clock
		ClockWrite 					: BOOL;				// (NA) Modbus writing Clock 	

    //M_CP VARIABLES//
		Trig_Cmd_Read						: R_TRIG;                                                                                        
		Trig_Cmd_Write						: R_TRIG;                                                                                        
	//M_INIT VARIABLES // 	        		
		bInit								: BOOL := TRUE ; 		// (NA) Initialize object parameters at first cycle 
				
END_VAR

METHOD M_AlarmManagement
//////////////////
// Manages Contactor alarms and warnings
/////////////////

VAR 
	// Method local variables (reinitialized at each cycle) 
	
END_VAR
END_METHOD

METHOD M_CP 
VAR_INPUT
END_VAR
END_METHOD

METHOD M_Execute
VAR_INPUT
END_VAR

VAR

END_VAR




// READING AND WRITING CLOCK //
	TP1(IN:=NOT TP1.Q , PT:= ParamClockReadTime);
	ClockRead 				:= TP1.Q;

	TP2(IN:=NOT TP2.Q , PT:= ParamClockWriteTime);
	ClockWrite 				:= TP2.Q;

// PERMANENT CONDITIONS //	
	
	
//Methods call	
	M_Read();
	M_Rotate(); 

	M_AlarmManagement();
END_METHOD

METHOD M_Read
//////////////////
// Manages Opening of the contactor
//////////////////

VAR 
	// Method local variables (reinitialized at each cycle) 
	KK: WORD ; 
	LL: WORD ; 
	JJ: WORD;
	MW: FB_MergeWordsToDint;
	MF : FB_MergeWordsToFloat ; 

	MesFlag				: ARRAY[1..5] OF  WORD;	
	MesAlarm2			: ARRAY[1..5] OF WORD;
	MesAlarm			: ARRAY[1..5] OF WORD;
	MesStatus			: ARRAY[1..5] OF WORD ; 
	MesStatusSynthesis	: WORD ; 

	CalTraNb: UINT;
END_VAR
END_METHOD

METHOD M_Rotate
//////////////////
// Manages Opening of the contactor
//////////////////

VAR 
	// Method local variables (reinitialized at each cycle) 

	CHECK: BOOL ;
	WriteCmd: BOOL ;
	CHECK1: BOOL ;
	WriteCmd1: BOOL ;	
	CHECK2: BOOL ;
	WriteCmd2: BOOL ;	
	CHECK3: BOOL ;
	WriteCmd3: BOOL ;	
		
	
	SetptGroupCmd		: WORD ; 




	FRS1: BOOL;

END_VAR
END_METHOD

END_FUNCTION_BLOCK

// ---- 01_Equipement_Library/Tracker/FB_NCU_Axial.TcPOU
FUNCTION_BLOCK  FB_NCU_Axial EXTENDS FB_NCU_Base
//////////////////
// NCU Function 
//////////////////
VAR_INPUT PERSISTENT
	// Parameters of the Object (instance/model specific) 

	                                                		
	ParamNbReadAtOnce			: BYTE:= 4 ; 				// Maximum 6	
	ParamTempoWindAlarm			: TIME 	:=T#10S		 ; 		// (s) Config : Tempo to detect Wind Alarm
END_VAR

VAR_INPUT 
	//Child objects
		IN_CmdEmergency 			: BOOL ; 				// (NA)  
		IN_CmdCleaning 				: BOOL ; 
		IN_CmdWind					: BOOL ; 
		IN_CmdSnow					: BOOL ; 
		IN_CmdReleaseAll			: BOOL; 
		IN_SetptGroupCmd			: WORD ; 
		MesDataExd						: NCU_Axial ; 
END_VAR


VAR
	//M_ROTATE VARIABLES//
		R_TRIG3					: R_TRIG;
		F_TRIG3					: F_TRIG;
		R_TRIG4					: R_TRIG;
		F_TRIG4					: F_TRIG;		
	
		R_TRIG2					: R_TRIG;
		F_TRIG2					: F_TRIG;
		R_TRIG1					: R_TRIG;
		F_TRIG1					: F_TRIG;
		
		RS1						: RS ; 
		RS2						: RS;
		RS3						: RS;		
		RS4						: RS;		
		
		
		MesForceWindCmd_save	: WORD;
		MesForceSnowCmd_save	: WORD;
		MesForceCleaning_save	: WORD ; 
		
		BlockWriteTemp		:ARRAY[1..4] OF WORD ; 

		
		
	//M_ALARMMANAGEMENT VARIABLES//

		TON_WindAlarm				: TON ;													// Tempo before detecting Wind Alarm. 
	
	
	
		
	//M_READ VARAIBLES 
		FB_ModbusRead	          	: ARRAY[1..6] OF  FB_ModbusRead; 	            // (NA) FB for Modbus Reading
		FB_ModbusRead_NCU          	: ARRAY[1..2] OF  FB_ModbusRead; 	            // (NA) FB for Modbus Reading
		FB_ModbusWrite				: ARRAY[1..4] OF FB_ModbusWrite;
		AX_ModbusReadAlarm			: ARRAY[1..6] OF BOOL;		
		AX_ModbusReadAlarmId		: ARRAY[1..6] OF UDINT;
		AX_ModbusReadAlarm_NCU		: ARRAY[1..2] OF BOOL;		
		AX_ModbusReadAlarmId_NCU	: ARRAY[1..2] OF UDINT;

	
		AX_ModbusWriteAlarm			: ARRAY[1..4] OF BOOL;
		AX_ModbusWriteAlarmId		: ARRAY[1..4] OF UDINT;
		
		
		MesBlock_Temp 				: ARRAY[1..6] OF  ARRAY [1..125] OF WORD ; 		// (NA) Temporary Block with multiple modbus reading (Caution : Double Word variables)	
		MesBlock_Temp_NCU			: ARRAY[1..2] OF ARRAY[1..125] OF WORD ; 
		
		CTU							: CTU ; 
		
	//M_STATEMANAGER VARIABLES//
	

		CalState					: BYTE ; 				// (NA) [P,H,B] Bit 0: Standby , Bit 1: Working 

		
	// M_EXECUTE VARIABLES 	//      
	
        
		CP_Rotate					: BOOL ; 				// (NA) Permanent Conditions
		CalCPEmergency					: BOOL ; 
		CalCPWindPos					: BOOL ;
		CalCPSnowPos					: BOOL ;
		CalCPCleaningPos				: BOOL ;

				
END_VAR

METHOD M_AlarmManagement
//////////////////
// Manages Contactor alarms and warnings
/////////////////

VAR 
	// Method local variables (reinitialized at each cycle) 
	FB_AlarmCodeManager			: FB_AlarmCodeManager ; 
	
	KK: INT;
	MesAlarmSynthesis: BOOL;
	MesBlockSynthesis: BOOL;

	ForceCmd: BOOL;
	ComWriteAlarm: BOOL;
	ComReadAlarm: BOOL;
	JJ: INT;
	bTest: BOOL;
END_VAR
// At lesat one tracker has an alarm 
MesAlarmSynthesis 	:=  TRUE  ;
MesBlockSynthesis 	:=  FALSE  ;

FOR KK:= 1 TO ParamNbTracker DO 
	MesAlarmSynthesis := MesAlarmSynthesis AND MesDataExd.AX_TRK[KK].MesStatusSynthesis.13 ; // At least one alarm is active	
	MesBlockSynthesis := MesBlockSynthesis OR MesDataExd.AX_TRK[KK].MesStatusSynthesis.14 ; // At least one tracker is blocked .  
END_FOR


ForceCmd := MesDataExd.MesForceCleaningCmd>0 OR  MesDataExd.MesForceSnowCmd>0 OR MesDataExd.MesForceWindCmd>0 ; // NCU is in force command


ComWriteAlarm :=AX_ModbusWriteAlarm[1] OR AX_ModbusWriteAlarm[2] OR AX_ModbusWriteAlarm[3] OR AX_ModbusWriteAlarm[4] ;  

ComReadAlarm := AX_ModbusReadAlarm_NCU[1] OR AX_ModbusReadAlarm_NCU[2]; 
FOR JJ:= 1 TO ParamNbReadAtOnce DO 
	ComReadAlarm :=  ComReadAlarm OR AX_ModbusReadAlarm[KK] ; 
END_FOR

TON_ComAlarm(IN:= ComReadAlarm, PT:= ParamTempoComAlarm, Q=>MesDataExd.MesData.MesAlarmCom) ;	
TON_WindAlarm(IN:=  MesDataExd.MesRSUGlobal.1, PT:= ParamTempoWindAlarm, Q=>MesDataExd.MesWindAlarm) ;

// ALARM CODE //
	FB_AlarmCodeManager(
		bAlarm1			:= MesAlarmSynthesis , 		// At least one tracker has a fault
		bAlarm2			:= MesBlockSynthesis , 		// At least one tracker is blocked
		bAlarm3			:= FALSE, 
		bAlarm4			:= FALSE,
		bAlarm5			:= FALSE,
		bAlarm6			:= MesDataExd.MesRSUGlobal.15,	// Flood Alarm
		bAlarm7			:= MesDataExd.MesRSUGlobal.6,	// Gust Wind NCU Alarm,	  	//,
		bAlarm8			:= MesDataExd.MesRSUGlobal.5,	// Snow  alarm,	  	//,
		bAlarm9			:= MEsDataExd.MesWindAlarm,	// Wind Alarm
		bAlarm10		:= FALSE,
		bAlarm11		:= FALSE,
		bAlarm12		:= FALSE,
		bAlarm13		:= FALSE,
		bAlarm14		:= FALSE,
		bAlarm15		:= ComWriteAlarm,
		wAlarmCode		=> MesDataExd.MesData.MesAlarmCode);
		

// WARNING CODE //
	FB_AlarmCodeManager(
 		bAlarm1			:= MesDataExd.MesComNCUAlarm>0 , // At least one NCU has a commuication alarm,		//
		bAlarm2			:= FALSE ,
		bAlarm3			:= MesDataExd.MesRSUGlobal.10,	// Flood Sensor communication alarm,	  	//
		bAlarm4			:= MesDataExd.MesRSUGlobal.9,	// Snow Sensor communication alarm,	  	//,		//
		bAlarm5			:= MesDataExd.MesRSUGlobal.8,	// Wind Sensor communication alarm,	  	//,		//
		bAlarm6			:= MesDataExd.MesRSUGlobal.0 , 		// Communication alarm with all RSUs . 
		bAlarm7			:= NOT MesAlarmSynthesis,		// at least on TCU has an alarm
		bAlarm8			:= MesBlockSynthesis,		// at least one tracker is blocked . ,       //
		bAlarm9			:= ForceCmd,       //	some TCU of the NCU are forced in a certain position
		bAlarm10		:= IN_CmdCleaning AND IN_CmdSnow OR IN_CmdCleaning AND IN_CmdWind OR IN_CmdSnow AND IN_CmdWind,       // Several commmands at the same time. 
		bAlarm11		:= FALSE,       //
		bAlarm12		:= FALSE,       //
		bAlarm13		:= FALSE, 
		bAlarm14		:= FALSE, 
		bAlarm15		:= MesDataExd.MesData.MesAlarmCom, 
		wAlarmCode		=> MesDataExd.MesData.MesWarningCode);	

	FB_AlarmCodeManager(
 		bAlarm1			:= IN_CmdCleaning, 
		bAlarm2			:= IN_CmdEmergency, 
		bAlarm3			:= IN_CmdSnow, 
		bAlarm4			:= IN_CmdWind, 
		bAlarm5			:= FALSE, 
		bAlarm6			:= FALSE, 
		bAlarm7			:= FALSE, 
		bAlarm8			:= FALSE, 
		bAlarm9			:= FALSE, 
		bAlarm10		:= FALSE, 
		bAlarm11		:= FALSE,       //
		bAlarm12		:= FALSE,       //
		bAlarm13		:= FALSE, 
		bAlarm14		:= FALSE, 
		bAlarm15		:= FALSE, 
		wAlarmCode		=> MesDataExd.MesData.MesEventCode);
END_METHOD

METHOD M_CP 
VAR_INPUT
END_VAR

SUPER^.M_CP() ; 




Trig_Cmd_Read(CLK:=IN_CmdToggleRead);
Trig_Cmd_Write(CLK:=IN_CmdToggleWrite);
	
IF Trig_Cmd_Read.Q THEN
	IN_CmdToggleRead := FALSE;
	MesDataExd.MesData.MesCP_Read := NOT MesDataExd.MesData.MesCP_Read;
END_IF


IF Trig_Cmd_Write.Q THEN
	IN_CmdToggleWrite := FALSE;
	MesDataExd.MesData.MesCP_Write := NOT MesDataExd.MesData.MesCP_Write;
END_IF



	CP_Rotate					:= NOT MesDataExd.MesData.MesAlarmCode.0 ; // No alarms on NCU

	CalCPEmergency				:= TRUE  ; //  CmdEmergency OR CmdWind OR CmdCleaning ; 
	                        	
	CalCPWindPos				:=NOT IN_CmdEmergency AND NOT IN_CmdSnow AND NOT IN_CmdCleaning AND NOT MesDataExd.MesData.MesAlarmCode.0  ; 
	CalCPSnowPos				:=NOT IN_CmdEmergency AND NOT IN_CmdWind AND NOT IN_CmdCleaning AND NOT MesDataExd.MesData.MesAlarmCode.0  ; 
	CalCPCleaningPos			:=NOT IN_CmdEmergency AND NOT IN_CmdWind AND NOT IN_CmdSnow AND NOT MesDataExd.MesData.MesAlarmCode.0 ; 
	
	
	MesDataExd.CalCPWindPos		:=CalCPWindPos		;
	MesDataExd.CalCPSnowPos		:=CalCPSnowPos		;
	MesDataExd.CalCPCleaningPos	:=CalCPCleaningPos	;
END_METHOD

METHOD M_Execute
VAR_INPUT
END_VAR

VAR

END_VAR

// READING AND WRITING CLOCK //
	TP1(IN:=NOT TP1.Q , PT:= ParamClockReadTime);
	ClockRead 				:= TP1.Q;

	TP2(IN:=NOT TP2.Q , PT:= ParamClockWriteTime);
	ClockWrite 				:= TP2.Q;

// PERMANENT CONDITIONS //	




	

	
//Methods call	
	M_Read();
	M_Rotate(); 

	M_AlarmManagement();
END_METHOD

METHOD M_Read
//////////////////
// Manages Opening of the contactor
//////////////////

VAR 
	// Method local variables (reinitialized at each cycle) 
	KK: WORD ; 
	LL: WORD ; 
	JJ: WORD;
	MW: FB_MergeWordsToDint;
	MF : FB_MergeWordsToFloat ; 

	MesFlag				: ARRAY[1..5] OF  WORD;	
	MesAlarm2			: ARRAY[1..5] OF WORD;
	MesAlarm			: ARRAY[1..5] OF WORD;
	MesStatus			: ARRAY[1..5] OF WORD ; 
	MesStatusSynthesis	: WORD ; 

	CalTraNb: UINT;
END_VAR

IF MesDataExd.MesData.MesCP_Read THEN 

	// READ NCU DAta 
		FB_ModbusRead_NCU[1]
		(
			nTCPPort	:= ParamTcpPort,
			ClockRead:= MesDataExd.MesData.MesCP_Read AND ClockRead, 
			Reset:= CmdClearFault_G,
			sIPAddr:=ParamIPAddress ,
			nUnitID:= 1, 
			tTimeout:= ParamTimeout,
			nQuantity		:= 125 , 
			nMBAddr			:=  30000, 
			cbLength		:= SIZEOF(MesBlock_Temp_NCU[1]) , 
			pDestAddr		:= ADR(MesBlock_Temp_NCU[1]) , 
			ModbusReadAlarm	=>AX_ModbusReadAlarm_NCU[1] , 
			ErrorId			=> AX_ModbusReadAlarmId_NCU[1]
		);
	
	
	MesDataExd.MesRSuGlobal:=MesBlock_Temp_NCU[1][3];
	//MesData.MesAnemoAlarm:=MesBlock_Temp_NCU[1][4];
	MesDataExd.MesComNCUAlarm:=MesBlock_Temp_NCU[1][37];
	MF( WORD_STRONG:= MesBlock_Temp_NCU[1][47],  WORD_WEAK := MesBlock_Temp_NCU[1][48],  VAR_OUT :=MesDataExd.MesWindSpeed);
	MF( WORD_STRONG:= MesBlock_Temp_NCU[1][67],  WORD_WEAK := MesBlock_Temp_NCU[1][68],  VAR_OUT:=MesDataExd.MesSnow);
	MF( WORD_STRONG:= MesBlock_Temp_NCU[1][107], WORD_WEAK := MesBlock_Temp_NCU[1][108], VAR_OUT:=MesDataExd.MesWindDir);
	
	
	// READ TCU DATA 
	CTU(CU:=ClockRead , PV:= REAL_TO_WORD(ParamNbTracker/(ParamNbReadAtOnce*5))+1 ) ; 
	CTU(RESET:= CTU.Q ) ; 
	LL:= (CTU.CV)  ; // At every Clock Read , we read a new 4 blocks of 5 trackers >> 20 trackers . We reset once all trackers have been read.  
	
	// MODBUS REQUEST//
		// Lecture de 4 block en meme temps modbus  
		//Chaque block contient les infos de 5 TCU 
		// A chaque clock read , 20 TCU sont lus . 
		// On fait une rotation 
	
	FOR KK := 1 TO ParamNbReadAtOnce DO 	
		FB_ModbusRead[KK]
		(
			nTCPPort	:= ParamTcpPort,
			ClockRead:= MesDataExd.MesData.MesCP_Read AND ClockRead, 
			Reset:= CmdClearFault_G,
			sIPAddr:=ParamIPAddress ,
			nUnitID:= 1, 
			tTimeout:= ParamTimeout,
			nQuantity		:= 110 , 
			nMBAddr			:= 30146 + (KK-1)*110 + (LL)*ParamNbReadAtOnce*110 , 
			cbLength		:= SIZEOF(MesBlock_Temp[KK]) , 
			pDestAddr		:= ADR(MesBlock_Temp[KK]) , 
			ModbusReadAlarm	=>AX_ModbusReadAlarm[KK] , 
			ErrorId			=> AX_ModbusReadAlarmId[KK]
		);
		
		CalTraNb := 5*ParamNbReadAtOnce*LL+5*(KK-1) ; 
		
		// Read 
			// TCU #1
			FOR JJ:= 1 TO 5 DO 
				CalTraNb := CalTraNb +1 ; 	
				IF CalTraNb > ParamNbTracker THEN 
					EXIT ; 
				END_IF
				MesStatus[JJ]	:=MesBlock_Temp[KK][2+22*(JJ-1)];
				MesAlarm[JJ]	:=MesBlock_Temp[KK][3+22*(JJ-1)];
				MesAlarm2[JJ]	:=MesBlock_Temp[KK][4+22*(JJ-1)];
				MesFlag[JJ]		:=MesBlock_Temp[KK][5+22*(JJ-1)];
				
				MF( WORD_STRONG:= MesBlock_Temp[KK][7+22*(JJ-1)], WORD_WEAK := MesBlock_Temp[KK][8+22*(JJ-1)], VAR_OUT:=MesDataExd.AX_TRK[CalTraNb].MesData.MesAngle);
				MW(WORD_STRONG:= MesBlock_Temp[KK][ 9+22*(JJ-1)], 	SIGNED:=TRUE, FIX:=3 , SIZE:=1, VAR_OUT:=MesDataExd.AX_TRK[CalTraNb].MesImotor);
				MW(WORD_STRONG:= MesBlock_Temp[KK][ 10+22*(JJ-1)], 	SIGNED:=TRUE, FIX:=3 , SIZE:=1, VAR_OUT:=MesDataExd.AX_TRK[CalTraNb].MesImaxmotor);
				MF( WORD_STRONG:= MesBlock_Temp[KK][11+22*(JJ-1)], WORD_WEAK := MesBlock_Temp[KK][12+22*(JJ-1)], VAR_OUT:=MesDataExd.AX_TRK[CalTraNb].MesData.MesAngleTarget);
			
				
				MesStatusSynthesis.0 := NOT(MesStatus[JJ].8) AND NOT(MesStatus[JJ].9) ; // OFF 
				MesStatusSynthesis.1 := NOT(MesStatus[JJ].8) AND MesStatus[JJ].9; // MANUAL
				MesStatusSynthesis.2 := MesStatus[JJ].8 AND NOT(MesStatus[JJ].9) ; // AUTO 
				MesStatusSynthesis.3 := MesStatus[JJ].12 ; 
				MesStatusSynthesis.4 := MesStatus[JJ].11 ; 
				MesStatusSynthesis.5 := MesStatus[JJ].0 ; 
				MesStatusSynthesis.6 := MesAlarm[JJ].8	; 
				MesStatusSynthesis.7 := MesAlarm[JJ].7; 
				MesStatusSynthesis.8 := MesAlarm[JJ].5 ; 
				MesStatusSynthesis.9 := MesAlarm[JJ].4 ; 
				MesStatusSynthesis.10:= MesAlarm2[JJ].14 ; 
				MesStatusSynthesis.11:= MesAlarm2[JJ].5 ; 
				MesStatusSynthesis.12:= MesAlarm2[JJ].4 ; 
				MesStatusSynthesis.13:= NOT MesFlag[JJ].15 ; // One alarm is active  
				MesStatusSynthesis.14:= MesFlag[JJ].11 ; 
				MesStatusSynthesis.15:= MesFlag[JJ].7 ; 
				
				MesDataExd.AX_TRK[CalTraNb].MesStatusSynthesis:= MesStatusSynthesis ; 
				// angle en degres. 
				MesDataExd.AX_TRK[CalTraNb].MesData.MesAngle:= MesDataExd.AX_TRK[CalTraNb].MesData.MesAngle * 360 / (2*PI) ; 
				MesDataExd.AX_TRK[CalTraNb].MesData.MesAngleTarget:= MesDataExd.AX_TRK[CalTraNb].MesData.MesAngleTarget * 360 / (2*PI) ;
			END_FOR
	
	END_FOR 


END_IF
END_METHOD

METHOD M_Rotate
//////////////////
// Manages Opening of the contactor
//////////////////

VAR 
	// Method local variables (reinitialized at each cycle) 

	CHECK: BOOL ;
	WriteCmd: BOOL ;
	CHECK1: BOOL ;
	WriteCmd1: BOOL ;	
	CHECK2: BOOL ;
	WriteCmd2: BOOL ;	
	CHECK3: BOOL ;
	WriteCmd3: BOOL ;	
		
	
	SetptGroupCmd		: WORD ; 




	FRS1: BOOL;

END_VAR

// Realease all 
IF IN_CmdReleaseAll THEN 
	MesForceWindCmd_save := 0 ; 
	MesForceSnowCmd_save := 0 ; 
	MesForceCleaning_save :=0 ; 
END_IF


// Protect 
SetptGroupCmd :=  IN_SetptGroupCmd AND NOT(MesDataExd.MesForceCleaningCmd OR MesDataExd.MesForceSnowCmd OR MesDataExd.MesForceWindCmd ) ; 

// READ Force Status 

	FB_ModbusRead_NCU[2]
	(
		nTCPPort	:= ParamTcpPort,
		ClockRead:= MesDataExd.MesData.MesCP_Read AND ClockRead, 
		Reset:= CmdClearFault_G,
		sIPAddr:=ParamIPAddress ,
		nUnitID:= 1, 
		tTimeout:= ParamTimeout,
		nQuantity		:= 3 , 
		nMBAddr			:=  50086, 
		cbLength		:= SIZEOF(MesBlock_Temp_NCU[2]) , 
		pDestAddr		:= ADR(MesBlock_Temp_NCU[2]) , 
		ModbusReadAlarm	=>AX_ModbusReadAlarm_NCU[2] , 
		ErrorId			=> AX_ModbusReadAlarmId_NCU[2]
	);

MesDataExd.MesForceWindCmd	:= MesBlock_Temp_NCU[2][1] ; 
MesDataExd.MesForceSnowCmd	:= MesBlock_Temp_NCU[2][2] ; 
MesDataExd.MesForceCleaningCmd := MesBlock_Temp_NCU[2][3] ; 


// EMERGENCY POSITION . 
// On regarde l'état de la variable forcée avant écriture que l'on mémorise . Une fois la commande d'urgence relachee, on retourne au même état que précédemment? 

BlockWriteTemp[1] := MesDataExd.MesForceWindCmd ; 

// On mémorise l'état d'avant commande 

R_TRIG1(CLK:=IN_CmdEmergency ) ; 
F_TRIG1(CLK:= IN_CmdEmergency ) ; 
IF R_TRIG1.Q AND NOT RS1.Q1 THEN 
	MesForceWindCmd_save	:= MesDataExd.MesForceWindCmd ; 
END_IF
// On reattribue la commande sauvegardée  et on la maintient jusqu'à ce que la commande soit passée 
RS1(SET:= F_TRIG1.Q , RESET1:=FB_ModbusWrite[1].Completed ); 
IF RS1.Q1 THEN 
	BlockWriteTemp[1] :=  MesForceWindCmd_save ; 
END_IF

IF IN_CmdEmergency THEN 
	BlockWriteTemp[1] := SEL(IN_CmdReleaseAll ,   2#1111111111  , 0) ; 

END_IF 
	

// WRITE ON CHANGE //
	// Detect if another status is already forced . 
	CHECK := BlockWriteTemp[1] <> MesDataExd.MesForceWindCmd ; 

	WriteCmd 			:=(CHECK AND  ClockWrite) AND CalCPEmergency; 
	
			FB_ModbusWrite[1]
		(
			pSrcAddr := ADR (BlockWriteTemp[1]),
			sIPAddr := ParamIPAddress,
			tTimeout := ParamTimeout,
			nMBAddr := 50086, // 
			nTCPport := ParamTCPPort,
			cbLength := SIZEOF(BlockWriteTemp[1]),
			nQuantity := 1,
			nUnitID := ParamUnitID,
			WriteCmd := WriteCmd AND MesDataExd.MesData.MesCP_Write,
			Reset := CmdClearFault_G ,
			ErrorId => AX_ModbusWriteAlarmId[1],
			ModbusWriteAlarm => AX_ModbusWriteAlarm[1]
		);
		
// WIND POSITION 
// On attribue la commande à ce qui est lu sur le registre pour ne pas écraser une commande reçue sauf si une écriture est en cours. 



BlockWriteTemp[2] := MesDataExd.MesForceWindCmd ; 



// On mémorise l'état d'avant commande 
R_TRIG2(CLK:=CalCPWindPos AND IN_CmdWind ) ; 
F_TRIG2(CLK:= CalCPWindPos AND IN_CmdWind ) ; 
IF R_TRIG2.Q AND NOT RS2.Q1 THEN 
	MesForceWindCmd_save	:= MesDataExd.MesForceWindCmd ; 
END_IF
// On reattribue la commande sauvegardée  et on la maintient jusqu'à ce que la commande soit passée 
RS2(SET:= F_TRIG2.Q , RESET1:=FB_ModbusWrite[2].Completed ) ; 
IF RS2.Q1 THEN 
	BlockWriteTemp[2] :=  MesForceWindCmd_save ; 
END_IF

IF CalCPWindPos AND IN_CmdWind AND (SetptGroupCmd<>0) THEN 
	BlockWriteTemp[2] :=  SetptGroupCmd OR MesForceWindCmd_save ; 

END_IF 
	
// WRITE ON CHANGE //
	// Detect if another status is already forced . 
	CHECK1 := BlockWriteTemp[2] <> MesDataExd.MesForceWindCmd ; 

	WriteCmd1 			:=(CHECK1 AND  ClockWrite) AND CalCPWindPos; 
	
			FB_ModbusWrite[2]
		(
			pSrcAddr := ADR (BlockWriteTemp[2]),
			sIPAddr := ParamIPAddress,
			tTimeout := ParamTimeout,
			nMBAddr := 50086, // 
			nTCPport := ParamTCPPort,
			cbLength := SIZEOF(BlockWriteTemp[2]),
			nQuantity := 1,
			nUnitID := ParamUnitID,
			WriteCmd := WriteCmd1 AND MesDataExd.MesData.MesCP_Write,
			Reset := CmdClearFault_G ,
			ErrorId => AX_ModbusWriteAlarmId[2],
			ModbusWriteAlarm => AX_ModbusWriteAlarm[2]
		);		
		
// SNOW  POSITION 
// On attribue la commande à ce qui est lu sur le registre pour ne pas écraser une commande reçue sauf si une écriture est en cours. 

BlockWriteTemp[3] := MesDataExd.MesForceSnowCmd ; 

// On mémorise l'état d'avant commande 
R_TRIG3(CLK:=CalCPSnowPos AND IN_CmdSnow ) ; 
F_TRIG3(CLK:= CalCPSnowPos AND IN_CmdSnow ) ; 
IF R_TRIG3.Q AND NOT RS3.Q1 THEN 
	MesForceSnowCmd_save	:= MesDataExd.MesForceSnowCmd ; 
END_IF
// On reattribue la commande sauvegardée  et on la maintient jusqu'à ce que la commande soit passée 
RS3(SET:= F_TRIG3.Q , RESET1:=FB_ModbusWrite[3].Completed ) ; 
IF RS3.Q1 THEN 
	BlockWriteTemp[3] :=  MesForceSnowCmd_save ; 
END_IF

IF CalCPSnowPos AND IN_CmdSnow AND (SetptGroupCmd<>0)THEN 
	BlockWriteTemp[3] :=  SetptGroupCmd OR MesForceSnowCmd_save ; 

END_IF 
	
// WRITE ON CHANGE //
	// Detect if another status is already forced . 
	CHECK2 := BlockWriteTemp[3] <> MesDataExd.MesForceSnowCmd ; 

	WriteCmd2 			:=(CHECK2 AND  ClockWrite) AND CalCPSnowPos; 
	
			FB_ModbusWrite[3]
		(
			pSrcAddr := ADR (BlockWriteTemp[3]),
			sIPAddr := ParamIPAddress,
			tTimeout := ParamTimeout,
			nMBAddr := 50087, // 
			nTCPport := ParamTCPPort,
			cbLength := SIZEOF(BlockWriteTemp[3]),
			nQuantity := 1,
			nUnitID := ParamUnitID,
			WriteCmd := WriteCmd2 AND MesDataExd.MesData.MesCP_Write,
			Reset := CmdClearFault_G ,
			ErrorId => AX_ModbusWriteAlarmId[3],
			ModbusWriteAlarm => AX_ModbusWriteAlarm[3]
		);		
				
// CLEANING  POSITION 
// On attribue la commande à ce qui est lu sur le registre pour ne pas écraser une commande reçue sauf si une écriture est en cours. 

BlockWriteTemp[4] := MesDataExd.MesForceCleaningCmd ; 

// On mémorise l'état d'avant commande 
R_TRIG4(CLK:=CalCPCleaningPos AND IN_CmdCleaning ) ; 
F_TRIG4(CLK:= CalCPCleaningPos AND IN_CmdCleaning ) ; 
IF R_TRIG4.Q AND NOT RS4.Q1 THEN 
	MesForceCleaning_save	:= MesDataExd.MesForceCleaningCmd ; 
END_IF
// On reattribue la commande sauvegardée  et on la maintient jusqu'à ce que la commande soit passée 
RS4(SET:= F_TRIG4.Q , RESET1:=FB_ModbusWrite[4].Completed) ; 
IF RS4.Q1 THEN 
	BlockWriteTemp[4] :=  MesForceCleaning_save ; 
END_IF

IF CalCPCleaningPos AND IN_CmdCleaning AND (SetptGroupCmd<>0) THEN 
	BlockWriteTemp[4] :=  SetptGroupCmd OR MesForceCleaning_save ; 

END_IF 
	
// WRITE ON CHANGE //
	// Detect if another status is already forced . 
	CHECK3 := BlockWriteTemp[4] <> MesDataExd.MesForceCleaningCmd ; 

	WriteCmd3 			:=(CHECK3 AND  ClockWrite) AND CalCPCleaningPos; 
	
			FB_ModbusWrite[4]
		(
			pSrcAddr := ADR (BlockWriteTemp[4]),
			sIPAddr := ParamIPAddress,
			tTimeout := ParamTimeout,
			nMBAddr := 50088, // 
			nTCPport := ParamTCPPort,
			cbLength := SIZEOF(BlockWriteTemp[4]),
			nQuantity := 1,
			nUnitID := ParamUnitID,
			WriteCmd := WriteCmd3 AND MesDataExd.MesData.MesCP_Write,
			Reset := CmdClearFault_G ,
			ErrorId => AX_ModbusWriteAlarmId[4],
			ModbusWriteAlarm => AX_ModbusWriteAlarm[4]
		);
END_METHOD

END_FUNCTION_BLOCK

// ---- 01_Equipement_Library/Transfo/FB_Transfo_Base.TcPOU
FUNCTION_BLOCK FB_Transfo_Base
//////////////////
// High Voltage transformer with Transfo or DMCR detection . 
//////////////////

VAR_INPUT PERSISTENT
	// Parameters of the Object (instance/model specific) 
	ParamTimeOut_Alarm   		    : TIME  := T#200MS  ;		(* (ms) Config : Tempo when open and close before raising alarm*)

END_VAR

VAR_OUTPUT
	//Child objects
	
END_VAR

VAR_INPUT
		// Transfo

END_VAR

VAR
	///MesDataExd					: Transfo ; 
		MesCP_Read					: BOOL := TRUE;	(* Read function enable *)
		MesCP_Write					: BOOL := TRUE;	(* Write function enable *)	
END_VAR

METHOD M_AlarmManagement
//////////////////
// Manages High Voltage Transformer Alarms
/////////////////

VAR 
	// Method local variables (reinitialized at each cycle) 
	FB_AlarmCodeManager : FB_AlarmCodeManager ; 

	
END_VAR
END_METHOD

METHOD M_Execute
//////////////////
//  Method Calls 
/////////////////

VAR 
	// Method local variables (reinitialized at each cycle) 

END_VAR

	
// METHODS CALLS //
	M_Read();
	M_AlarmManagement();
END_METHOD

METHOD M_Read : BOOL
VAR_INPUT
END_VAR

VAR
	MesAuxTransfoGazDischarge: INT;
	MesAuxTransfoTempTrigger: INT;
END_VAR
END_METHOD

END_FUNCTION_BLOCK

// ---- 01_Equipement_Library/Transfo/FB_Transfo_HVCom.TcPOU
FUNCTION_BLOCK FB_Transfo_HVCom EXTENDS FB_Transfo_Base
//////////////////
// High Voltage transformer with Transfo or DMCR detection . 
//////////////////

VAR_INPUT PERSISTENT
	// Parameters of the Object (instance/model specific) 
	
END_VAR

VAR_OUTPUT
	//Child objects
	
END_VAR

VAR_INPUT
MesDataExd		AT %Q*			: Transfo_HV ; 
		
END_VAR

VAR

END_VAR

METHOD M_AlarmManagement
//////////////////
// Manages High Voltage Transformer Alarms
/////////////////

VAR 
	// Method local variables (reinitialized at each cycle) 
	FB_AlarmCodeManager : FB_AlarmCodeManager ; 

	
END_VAR



// ALARM CODE //
	FB_AlarmCodeManager(
		bAlarm1			:= MesDataExd.MesData.MesAlarmTemp ,				// Temperature Alarm
		bAlarm2			:= MesDataExd.MesData.MesAlarmGas  , 				// Gas Alarm
		bAlarm3			:= MesDataExd.MesData.MesAlarmOilLevel  , 			// Pressure Alarm
		bAlarm4			:= FALSE, 								//
		bAlarm5			:= FALSE, 								//
		bAlarm6			:= FALSE,                               //
		bAlarm7			:= FALSE,                               //
		bAlarm8			:= FALSE,                               //
		bAlarm9			:= FALSE, 								//
		bAlarm10		:= FALSE,                               //
		bAlarm11		:= FALSE,                               //
		bAlarm12		:= FALSE,                               //
		bAlarm13		:= FALSE, 								//
		bAlarm14		:= FALSE,                               //
		bAlarm15		:= FALSE , 								//      
		wAlarmCode		=>MesDataExd.MesData.MesAlarmCode);               

// WARNING CODE //
	FB_AlarmCodeManager(
		bAlarm1 		:= FALSE,   							//
		bAlarm2			:= FALSE, 		                   	 	//
		bAlarm3			:= FALSE, 		                      	//
		bAlarm4			:= FALSE, 		                    	//
		bAlarm5			:= FALSE,                               //
		bAlarm6			:= FALSE,                               //
		bAlarm7			:= FALSE,                               //
		bAlarm8			:= FALSE,                               //
		bAlarm9			:= FALSE,                               //
		bAlarm10		:= FALSE,                               //
		bAlarm11		:= FALSE,                               //
		bAlarm12		:= FALSE,                               //
		bAlarm13		:= FALSE,                               //
		bAlarm14		:= FALSE,                               //
		bAlarm15		:= FALSE,                               //
		wAlarmCode		=>MesDataExd.MesData.MesWarningCode);
		
// EVENT CODE //
	FB_AlarmCodeManager(
		bAlarm1			:= FALSE, 			// 
		bAlarm2			:= FALSE, 			// 
		bAlarm3			:= FALSE, 			// 
		bAlarm4			:= FALSE, 			// 
		bAlarm5			:= FALSE,         	//
		bAlarm6			:= FALSE,         	//
		bAlarm7			:= FALSE,         	//
		bAlarm8			:= FALSE,         	//
		bAlarm9			:= FALSE,         	//
		bAlarm10		:= FALSE,         	//
		bAlarm11		:= FALSE,         	//
		bAlarm12		:= FALSE,         	//
		bAlarm13		:= FALSE,         	//
		bAlarm14		:= FALSE,         	//
		bAlarm15		:= FALSE,         	//
		wAlarmCode		=>MesDataExd.MesData.MesEventCode);
END_METHOD

METHOD M_Read : BOOL
VAR_INPUT
END_VAR

VAR
	MesAuxTransfoGazDischarge: INT;
	MesAuxTransfoTempTrigger: INT;
END_VAR
END_METHOD

END_FUNCTION_BLOCK

// ---- 01_Equipement_Library/Transfo/FB_Transfo_MV.TcPOU
FUNCTION_BLOCK FB_Transfo_MV EXTENDS FB_Transfo_Base
//////////////////
// High Voltage transformer with DGPT2 detection . 
//////////////////

VAR_INPUT PERSISTENT
	
	// Parameters of the Object (instance/model specific) 
	
		ParamNC					: BOOL  ; 			(* Normally closed inputs . If TRUE , 1 =  no alarms. *)
		
END_VAR

VAR_OUTPUT
	//Child objects
	
END_VAR

VAR_INPUT
	
	// Transfo
	
		IN_MesWarningTemp_IO				: BOOL ; 		// (NA) Oil Temperature Warning IO
		IN_MesAlarmTemp_IO					: BOOL ; 		// (NA) Oil Temperature Alarm IO
		IN_MesAlarmGas_IO					: BOOL ; 		// (NA) Gas Alarm IO
		IN_MesAlarmPressure_IO				: BOOL ; 		// (NA) Pressure Alarm IO
		IN_MesAlarmsSynthesis_IO			: BOOL ;        // (NA) Synthesis Alarms  IO 
		IN_MesAlarmOilLevel_IO				: BOOL ;		// (NA) Oil level Alarm IO
		IN_MesAlarmPowerSupply_IO			: BOOL ;		// (NA) Power Supply Alarm IO
	
		MesDataExd				   			: Transfo_MV ; 
	
END_VAR

VAR
	
	// Transfo
	
		TP_AlarmTemp 			: TP ;		
		TP_AlarmGas   		    : TP ;
		TP_AlarmOilLevel   		: TP ;
		TP_AlarmsSynthesis 		: TP ;
		TP_WarningTemp   	    : TP ;
		TP_AlarmPressure		: TP ;
		TP_AlarmPowerSupply		: TP ;

END_VAR

METHOD M_AlarmManagement
//////////////////
// Manages High Voltage Transformer Alarms
/////////////////

VAR 
	// Method local variables (reinitialized at each cycle) 
	FB_AlarmCodeManager : FB_AlarmCodeManager ; 

	
END_VAR
IF ParamNC THEN 
	
	MesDataExd.MesData.MesAlarmPowerSupply		:= NOT IN_MesAlarmPowerSupply_IO ; 
	MesDataExd.MesData.MesAlarmsSynthesis		:= NOT IN_MesAlarmsSynthesis_IO ; 
	MesDataExd.MesData.MesAlarmGas				:= NOT IN_MesAlarmGas_IO ; 
	MesDataExd.MesData.MesAlarmOilLevel 		:= NOT IN_MesAlarmOilLevel_IO ; 
	MesDataExd.MesData.MesAlarmTemp				:= NOT IN_MesAlarmTemp_IO ; 
	MesDataExd.MesData.MesWarningTemp			:= NOT  IN_MesWarningTemp_IO ;
	MesDataExd.MesData.MesAlarmPressure			:= NOT IN_MesAlarmPressure_IO ; 
	
ELSE
	
	MesDataExd.MesData.MesAlarmPowerSupply		:= IN_MesAlarmPowerSupply_IO ; 
	MesDataExd.MesData.MesAlarmsSynthesis		:= IN_MesAlarmsSynthesis_IO ; 
	MesDataExd.MesData.MesAlarmGas				:= IN_MesAlarmGas_IO ; 
	MesDataExd.MesData.MesAlarmOilLevel 		:= IN_MesAlarmOilLevel_IO ; 
	MesDataExd.MesData.MesAlarmTemp				:= IN_MesAlarmTemp_IO ;  
	MesDataExd.MesData.MesWarningTemp			:= IN_MesWarningTemp_IO ; 
	MesDataExd.MesData.MesAlarmPressure			:= IN_MesAlarmPressure_IO ;

END_IF



TP_AlarmTemp 		  (	IN:=NOT MesDataExd.MesData.MesAlarmTemp 	   	,PT := ParamTimeOut_Alarm  );
TP_AlarmGas   		  (	IN:=NOT MesDataExd.MesData.MesAlarmGas   	  	,PT := ParamTimeOut_Alarm  );
TP_AlarmOilLevel      (	IN:=NOT MesDataExd.MesData.MesAlarmOilLevel  	,PT := ParamTimeOut_Alarm  );
TP_AlarmsSynthesis    (	IN:=NOT MesDataExd.MesData.MesAlarmsSynthesis	,PT := ParamTimeOut_Alarm  );
TP_WarningTemp   	  (	IN:=NOT MesDataExd.MesData.MesWarningTemp   	,PT := ParamTimeOut_Alarm  );
TP_AlarmPowerSupply   (	IN:=NOT MesDataExd.MesData.MesAlarmPowerSupply  ,PT := ParamTimeOut_Alarm  );
TP_AlarmPressure	  (	IN:=NOT MesDataExd.MesData.MesAlarmPressure     ,PT := ParamTimeOut_Alarm  );

// ALARM CODE //
	FB_AlarmCodeManager(
		bAlarm1			:= MesDataExd.MesData.MesAlarmTemp ,				// Transfo Temperature Alarm
		bAlarm2			:= MesDataExd.MesData.MesAlarmGas  , 				// Transfo Gas Alarm
		bAlarm3			:= MesDataExd.MesData.MesAlarmOilLevel  , 			// Transfo Oil Level Alarm	
		bAlarm4			:= MesDataExd.MesData.MesAlarmsSynthesis, 			// Transfo Synthesis Alarm 
		bAlarm5			:= MesDataExd.MesData.MesAlarmPowerSupply ,			// Transfo Power Supply Alarm             
		bAlarm6			:= MesDataExd.MesData.MesAlarmPressure ,            // Pressure Alarm              
		bAlarm7			:= FALSE ,//            
		bAlarm8			:= FALSE ,//
		bAlarm9			:= FALSE, 								//
		bAlarm10		:= FALSE,                               //
		bAlarm11		:= FALSE,                               //
		bAlarm12		:= FALSE,                               //
		bAlarm13		:= FALSE, 								//
		bAlarm14		:= FALSE,                               //
		bAlarm15		:= FALSE , 								//      
		wAlarmCode		=>MesDataExd.MesData.MesAlarmCode);               

// WARNING CODE //
	FB_AlarmCodeManager(
		bAlarm1 		:= MesDataExd.MesData.MesWarningTemp,   			// Transfo Temperature Warning
		bAlarm2			:= FALSE ,//
		bAlarm3			:= FALSE, 		                      	//
		bAlarm4			:= FALSE, 		                    	//
		bAlarm5			:= FALSE,                               //
		bAlarm6			:= FALSE,                               //
		bAlarm7			:= FALSE,                               //
		bAlarm8			:= FALSE,                               //
		bAlarm9			:= FALSE,                               //
		bAlarm10		:= FALSE,                               //
		bAlarm11		:= FALSE,                               //
		bAlarm12		:= FALSE,                               //
		bAlarm13		:= FALSE,                               //
		bAlarm14		:= FALSE,                               //
		bAlarm15		:= FALSE,                               //
		wAlarmCode		=>MesDataExd.MesData.MesWarningCode);
		
// EVENT CODE //
	FB_AlarmCodeManager(
		bAlarm1			:= TP_AlarmTemp.Q ,						// Transfo Temperature Alarm back to normal             
		bAlarm2			:= TP_AlarmGas .Q ,						// Transfo Gas Alarm back to normal                   
		bAlarm3			:= TP_AlarmOilLevel.Q ,					// Transfo Oil Level Alarm back to normal     
		bAlarm4			:= TP_AlarmsSynthesis.Q ,				// Transfo Synthesis Alarm back to normal          
		bAlarm5			:= TP_WarningTemp.Q ,					// Transfo Temperature Warning back to normal 
		bAlarm6			:= TP_AlarmPowerSupply.Q ,				// Transfo Power Supply Alarm back to normal  
		bAlarm7			:= FALSE,         	//
		bAlarm8			:= FALSE,         	//
		bAlarm9			:= FALSE,         	//
		bAlarm10		:= FALSE,         	//
		bAlarm11		:= FALSE,         	//
		bAlarm12		:= FALSE,         	//
		bAlarm13		:= FALSE,         	//
		bAlarm14		:= FALSE,         	//
		bAlarm15		:= FALSE,         	//
		wAlarmCode		=>MesDataExd.MesData.MesEventCode);
END_METHOD

END_FUNCTION_BLOCK

// ---- 01_Equipement_Library/Transfo/FB_Transfo_MVCom.TcPOU
FUNCTION_BLOCK FB_Transfo_MVCom EXTENDS FB_Transfo_Base

//////////////////
// High Voltage transformer with Transfo or DMCR detection 
//////////////////

VAR_INPUT PERSISTENT
	// Parameters of the Object (instance/model specific) 
	
END_VAR

VAR_OUTPUT
	//Child objects
	
END_VAR

VAR_INPUT

	MesDataExd	AT %Q*				: Transfo_MV ; 
	
END_VAR

VAR
	
END_VAR

METHOD M_AlarmManagement
//////////////////
// Manages High Voltage Transformer Alarms
/////////////////

VAR 
	// Method local variables (reinitialized at each cycle) 
	FB_AlarmCodeManager : FB_AlarmCodeManager ; 

	
END_VAR
// ALARM CODE //
	FB_AlarmCodeManager(
		bAlarm1			:= MesDataExd.MesData.MesAlarmTemp  ,				// Temperature Alarm
		bAlarm2			:= MesDataExd.MesData.MesAlarmGas  , 				// Gas Alarm
		bAlarm3			:= MesDataExd.MesData.MesAlarmOilLevel  , 			// Oil Level Alarm
		bAlarm4			:= FALSE, 								//
		bAlarm5			:= FALSE, 								//
		bAlarm6			:= FALSE,                               //
		bAlarm7			:= FALSE,                               //
		bAlarm8			:= FALSE,                               //
		bAlarm9			:= FALSE, 								//
		bAlarm10		:= FALSE,                               //
		bAlarm11		:= FALSE,                               //
		bAlarm12		:= FALSE,                               //
		bAlarm13		:= FALSE, 								//
		bAlarm14		:= FALSE,                               //
		bAlarm15		:= FALSE , 								//      
		wAlarmCode		=>MesDataExd.MesData.MesAlarmCode);               

// WARNING CODE //
	FB_AlarmCodeManager(
		bAlarm1 		:= FALSE,   							//
		bAlarm2			:= FALSE, 		                   	 	//
		bAlarm3			:= FALSE, 		                      	//
		bAlarm4			:= FALSE, 		                    	//
		bAlarm5			:= FALSE,                               //
		bAlarm6			:= FALSE,                               //
		bAlarm7			:= FALSE,                               //
		bAlarm8			:= FALSE,                               //
		bAlarm9			:= FALSE,                               //
		bAlarm10		:= FALSE,                               //
		bAlarm11		:= FALSE,                               //
		bAlarm12		:= FALSE,                               //
		bAlarm13		:= FALSE,                               //
		bAlarm14		:= FALSE,                               //
		bAlarm15		:= FALSE,                               //
		wAlarmCode		=>MesDataExd.MesData.MesWarningCode);
		
// EVENT CODE //
	FB_AlarmCodeManager(
		bAlarm1			:= FALSE, 			// 
		bAlarm2			:= FALSE, 			// 
		bAlarm3			:= FALSE, 			// 
		bAlarm4			:= FALSE, 			// 
		bAlarm5			:= FALSE,         	//
		bAlarm6			:= FALSE,         	//
		bAlarm7			:= FALSE,         	//
		bAlarm8			:= FALSE,         	//
		bAlarm9			:= FALSE,         	//
		bAlarm10		:= FALSE,         	//
		bAlarm11		:= FALSE,         	//
		bAlarm12		:= FALSE,         	//
		bAlarm13		:= FALSE,         	//
		bAlarm14		:= FALSE,         	//
		bAlarm15		:= FALSE,         	//
		wAlarmCode		=>MesDataExd.MesData.MesEventCode);
END_METHOD

METHOD M_Read : BOOL
VAR_INPUT
END_VAR

VAR
	MesAuxTransfoGazDischarge: INT;
	MesAuxTransfoTempTrigger: INT;
END_VAR
END_METHOD

END_FUNCTION_BLOCK

// ---- 01_Equipement_Library/UPS/FB_UPS_MCSU4.TcPOU
FUNCTION_BLOCK FB_UPS_MCSU4 EXTENDS FB_UPS_Base
//////////////////
// UPS 
//////////////////
VAR_INPUT PERSISTENT
	// Parameters of the Object (instance/model specific) 
		ParamIPAddress				: STRING 	:= '192.168.20.66'; 	// (NA)Config: IP Adress of PV INverter
		ParamUnitID 				: BYTE  	:= 1; 			  		// (NA)   Modbus Unit ID. 
		ParamTCPPort				: UINT		:= 502;					// (NA) TCP port for modbus
		
END_VAR

VAR_OUTPUT
	//Child objects
	
END_VAR

VAR_INPUT
	IN_SwitchPos_IO					: BOOL; // Definition to be clarified during FAT	
	IN_MesBatHigh_IO		   		: BOOL;
	IN_RectifFail_IO				: BOOL;
		MesDataExd			AT %Q*	: UPS_MCSU4 ; 	
END_VAR

VAR
	//M_ALARMMANAGEMENT VARIABLES//

	//M_READ//

		AX_ModbusRead		   		: ARRAY [1..2] OF FB_ModbusRead ; 					// (NA) FB for Modbus Reading
		ModbusReadInput				: FB_ModbusReadInput ; 		       
                                 
		MesBlock_Temp 				: ARRAY [1..2] OF ARRAY[1..120]  OF WORD; 			// (NA) Temporary Block with multiple modbus reading (Caution : Double Word variables)
		MesBlockInput				: ARRAY[1..1] OF BYTE ; 
		
END_VAR

METHOD M_AlarmManagement
//////////////////
// Manages Rectifier Technologies UPS controller reference: MCSU4-HV.
/////////////////

VAR 
	// Method local variables (reinitialized at each cycle) 
	FB_AlarmCodeManager 	: FB_AlarmCodeManager ; 
END_VAR
	//Alarm	
	TON_ComAlarm	(IN:= (AX_ModbusRead[1].ModbusReadAlarm) AND (AX_ModbusRead[2].ModbusReadAlarm) AND (ModbusReadInput.ModbusReadAlarm) , PT:= ParamTempoComAlarm, 	Q=>MesDataExd.MesData.MesAlarmCom) ;	
	TON_ComWarning	(IN:= (AX_ModbusRead[1].ModbusReadAlarm) OR  (AX_ModbusRead[2].ModbusReadAlarm) OR  (ModbusReadInput.ModbusReadAlarm) , PT:= ParamTempoComWarning, 	Q=>MesWarningCom) ;	

	MesDataExd.MesAlarmUmax 	:= IN_MesBatHigh_IO;
	MesDataExd.MesAlarmRectifer := IN_RectifFail_IO;
	MesDataExd.MesOpen_CBBat 	:= A1_SUBMV.A1_UPS_24v.IN_SwitchPos_IO;
	
// ALARM CODE //
	FB_AlarmCodeManager(
		bAlarm1				:= MesDataExd.MesAlarmUmax, 				 				// Battery over voltage 
		bAlarm2				:= MesDataExd.MesData.MesAlarm_Ulow,						// Battery under voltage  
		bAlarm3				:= MesDataExd.MesData.MesAlarmState,						// UPS Fault synthesis
		bAlarm4				:= MesDataExd.MesOpen_CBBat, 								// CB battery Open  
		bAlarm5				:= MesDataExd.MesFuse_Burned,                               // Power distribution unit fuse fail
		bAlarm6				:= MesDataExd.MesAlarmRectifer, 							// Rectifier failure
		bAlarm7				:= FALSE, 													//
		bAlarm8				:= FALSE,                                                   //
		bAlarm9				:= FALSE,                                                   //
		bAlarm10			:= FALSE,                                                   //
		bAlarm11			:= FALSE,                                                   //
		bAlarm12			:= FALSE,                                                   //
		bAlarm13			:= FALSE,                                                   //
		bAlarm14			:= FALSE,                                                   //
		bAlarm15			:= FALSE , 													//
		wAlarmCode			=> MesDataExd.MesData.MesAlarmCode);

// WARNING CODE //
	FB_AlarmCodeManager(
		bAlarm1			:= MesDataExd.MesData.MesDischarging, 				 			// UPS discharging   														// 
		bAlarm2			:= MesDataExd.MesAlarmTemp_Bat,    								// Battery over temperature
		bAlarm3			:= MesWarningCom, 												// Communication warning  #COM
		bAlarm4			:= MesDataExd.MesData.MesAlarmCom,         						// Communication alarm    #COM													// 
		bAlarm5			:= MesDataExd.MesAlarmI_diff, 									//
		bAlarm6			:= MesDataExd.MesAlarmI_Earth,                                  //
		bAlarm7			:= FALSE,														//
		bAlarm8			:= MesDataExd.MesOpen_Aux,                                      // UPS auxiliary contacts open 
		bAlarm9			:= MesDataExd.MesAlarmTemp,         							// UPS over temperature
		bAlarm10		:= FALSE,                                                       //
		bAlarm11		:= FALSE,                                                       //
		bAlarm12		:= FALSE,                                                       //
		bAlarm13		:= FALSE,                                                       //
		bAlarm14		:= FALSE,                                                       //
		bAlarm15		:= FALSE,                                                       //
		wAlarmCode		=> MesDataExd.MesData.MesWarningCode);

// EVENT CODE //
	FB_AlarmCodeManager(
		bAlarm1			:=FALSE, 													// 
		bAlarm2			:=FALSE, 													// 
		bAlarm3			:=FALSE, 													// 
		bAlarm4			:=FALSE, 													// 
		bAlarm5			:=FALSE, 													//
		bAlarm6			:=FALSE,        											//
		bAlarm7			:=FALSE,        											//
		bAlarm8			:=FALSE,        											//
		bAlarm9			:=FALSE,        											//
		bAlarm10		:=FALSE,        											//
		bAlarm11		:=FALSE,        											//
		bAlarm12		:=FALSE,        											//
		bAlarm13		:=FALSE,        											//
		bAlarm14		:=FALSE,        											//
		bAlarm15		:=FALSE,        											//
		wAlarmCode		=> MesDataExd.MesData.MesEventCode);
END_METHOD

METHOD M_Read
//////////////////
//  Read Modbus Variable for UPS Rectifier Technologies MCSU4-HV. 
/////////////////
VAR 
	// Method local variables (reinitialized at each cycle) 	
		AX_Addr				: ARRAY[1..3] OF UINT := [16#82, 	16#C2, 	16#101];
		AX_Qty				: ARRAY[1..3] OF UINT := [16   ,	6 	 ,	4	  ];
		
		MW 					: FB_MergeWordsToDint; 
END_VAR


////////////////////// TO DO ///////////////
//MesDataExd.MesData := MesData ; // Allow to initialize MesData with code from UPS_Base ; 

IF MesDataExd.MesData.MesCP_Read THEN	

AX_ModbusRead[1]
(
	pDestAddr 		:= ADR(MesBlock_Temp[1]),
	sIPAddr 		:= ParamIPAddress,
	tTimeout 		:= ParamTimeout,
	nQuantity 		:= AX_Qty[1],
	ntcpport 		:= ParamTCPPort,
	nMBAddr 		:= AX_Addr[1]-2,
	nUnitID 		:= ParamUnitID,
	cbLength 		:= SIZEOF(MesBlock_Temp[1]),
	ClockRead 		:= ClockRead AND MesDataExd.MesData.MesCP_Read,
	Reset 			:= CmdClearFault_G OR IN_CmdReset_L,
);

AX_ModbusRead[2]
(
	pDestAddr 		:= ADR(MesBlock_Temp[2]),
	sIPAddr 		:= ParamIPAddress,
	tTimeout 		:= ParamTimeout,
	nQuantity 		:= AX_Qty[2],
	ntcpport 		:= ParamTCPPort,
	nMBAddr 		:= AX_Addr[2]-2,
	nUnitID 		:= ParamUnitID,
	cbLength 		:= SIZEOF(MesBlock_Temp[2]),
	ClockRead 		:= ClockRead AND MesDataExd.MesData.MesCP_Read,
	Reset 			:= CmdClearFault_G OR IN_CmdReset_L
);


ModbusReadInput
(
	pDestAddr 		:= ADR(MesBlockInput),
	sIPAddr 		:= ParamIPAddress,
	tTimeout 		:= ParamTimeout,
	nQuantity 		:= AX_Qty[3],
	ntcpport 		:= ParamTCPPort,
	nMBAddr 		:= AX_Addr[3]-1,
	nUnitID 		:= ParamUnitID,
	cbLength 		:= SIZEOF(MesBlockInput),
	ClockRead 		:= ClockRead AND MesDataExd.MesData.MesCP_Read,
	Reset 			:= GVL_CFG.CmdClearFault_G OR IN_CmdReset_L
);

//MW(WORD_STRONG:= MesBlock_Temp[1][3], WORD_WEAK := MesBlock_Temp[1][4],SIGNED:=TRUE, FIX:=2 , SIZE:=2, VAR_OUT:=MesDataExd.MesIload);
//MW(WORD_STRONG:= MesBlock_Temp[1][5], WORD_WEAK := MesBlock_Temp[1][6],SIGNED:=TRUE, FIX:=2 , SIZE:=2, VAR_OUT:=MesDataExd.MesUBatt);
//MW(WORD_STRONG:= MesBlock_Temp[1][7], WORD_WEAK := MesBlock_Temp[1][8],SIGNED:=TRUE, FIX:=2 , SIZE:=2, VAR_OUT:=MesDataExd.MesIBatt);
//MW(WORD_STRONG:= MesBlock_Temp[1][15], WORD_WEAK := MesBlock_Temp[1][16],SIGNED:=TRUE, FIX:=2 , SIZE:=2, VAR_OUT:=MesDataExd.MesSoC);
//
//MW(WORD_STRONG:= MesBlock_Temp[2][1], WORD_WEAK := MesBlock_Temp[2][2],SIGNED:=TRUE, FIX:=2 , SIZE:=2, VAR_OUT:=MesDataExd.MesIdc);
//MW(WORD_STRONG:= MesBlock_Temp[2][3], WORD_WEAK := MesBlock_Temp[2][4],SIGNED:=TRUE, FIX:=2 , SIZE:=2, VAR_OUT:=MesDataExd.MesData.MesUdc);
//MW(WORD_STRONG:= MesBlock_Temp[2][5], WORD_WEAK := MesBlock_Temp[2][6],SIGNED:=TRUE, FIX:=2 , SIZE:=2, VAR_OUT:=MesDataExd.MesU);
//
//MesDataExd.MesData.MesAlarm_Ulow := MesBlockInput[1].1	; // Low battery capacity 
//MesDataExd.MesOverTempBatt	:= MesBlockInput[1].2 ; // OverTemp battery 
//MesDataExd.MesData.MesDischarging := MesBlockInput[1].3 OR IN_MesDischarging_IO ; 
//MesDataExd.MesData.MesAlarmState := IN_MesFault_IO ; 
END_IF

//IF ParamNC THEN
//	MesDataExd.MesCBUpsOpened := IN_MesCbUPS_IO ; 
//	
//ELSE 
// 	MesDataExd.MesCBUpsOpened := NOT IN_MesCbUPS_IO ;
//END_IF
END_METHOD

END_FUNCTION_BLOCK

// ---- 01_Equipement_Library/UPS/FB_UPS_Base.TcPOU
FUNCTION_BLOCK FB_UPS_Base
//////////////////
// UPS 
//////////////////
VAR_INPUT PERSISTENT
	// Parameters of the Object (instance/model specific) 
		ParamTimeOut					: TIME := T#2S;		(* (s) Modbus Timeout*)
		ParamClockReadTime				: TIME := T#1S;		(* (s) Modbus Reading Frequency *)
		ParamNC							: BOOL := FALSE; 	(* (NA)False: TRUE = Closed, True : TRUE = opened*)
		                                
		ParamTempoComAlarm				: TIME := T#2S;		(* (s) Tempo before raising a communication alarm*)
		ParamTempoComWarning			: TIME := T#1S;		(* (s) Tempo before raising a communication warning*)
		ParamTP_Impulsion				: TIME := T#5S;		(* (s) TP Impulsion = 5s *)
END_VAR                                 
                                        
VAR_OUTPUT                              
	//Child objects                     
		OUT_CmdRelance_IO				: BOOL;
END_VAR                                 
                                        
VAR_INPUT                               
	// I/O Inputs                       
		IN_MesDischarging_IO		  	: BOOL;
		IN_MesBatLow_IO		   			: BOOL;
		IN_MesFault_IO					: BOOL;

		IN_CmdReStartUPS				: BOOL;
		
		IN_CmdToggleRead				: BOOL;
		IN_CmdReset_L					: BOOL; 
END_VAR

VAR
	//M_ALARMMANAGEMENT VARIABLES//
		TON_ComAlarm					: TON;
		TON_ComWarning					: TON;	

		MesWarningCom					: BOOL ; 			// (NA) [P,H] True if bad modbus communication 
			
	//M_READ//
//	MesDataExd					: UPS ; 

	//M_EXECUTE //
		TP1								: TP;
		ClockRead			AT %Q*		: BOOL;
   		
    //M_CP VARIABLES//
		Trig_Cmd_Read					: R_TRIG;                                                                                        
                                                                                       
		CmdRelanceChargeur				: BOOL;
		CP_Relance						: BOOL;
		TP_Relance						: TP;
		MesCP_Read					: BOOL := TRUE;	(* Read function enable *)
		MesCP_Write					: BOOL := TRUE;	(* Write function enable *)   
END_VAR

METHOD M_AlarmManagement
//////////////////
// Manages Sepam Alarms. Alarms opens HT CB until Sepam manual Reset . Warning Opens CB-L but does not maintain warning
/////////////////

VAR 
	// Method local variables (reinitialized at each cycle) 
	FB_AlarmCodeManager 	: FB_AlarmCodeManager ; 

 
END_VAR
END_METHOD

METHOD M_Execute
//////////////////
//  Method Calls 
/////////////////

VAR 
	// Method local variables (reinitialized at each cycle) 

END_VAR


// METHODS CALLS // 
CP_Relance	:= IN_CmdReStartUPS ; 	


	TP1(IN:=NOT TP1.Q , PT:= ParamClockReadTime);
	ClockRead 		:= TP1.Q;

	TP_Relance(IN:= CP_Relance , PT:=ParamTP_Impulsion) ;
	OUT_CmdRelance_IO	 := TP_Relance.Q ;
	
	M_Read(); 
	M_AlarmManagement() ;
END_METHOD

METHOD M_Read
//////////////////
//  Read Modbus Variable for PCS . 
/////////////////
VAR 
	// Method local variables (reinitialized at each cycle) 
		

END_VAR
END_METHOD

END_FUNCTION_BLOCK

// ---- 01_Equipement_Library/UPS/FB_UPS_PS10048.TcPOU
FUNCTION_BLOCK FB_UPS_PS10048 EXTENDS FB_UPS_Base
//////////////////
// SEPAM system for High Voltage or Low Voltage Grid Protection. 
//////////////////

VAR_INPUT 
	ParamTcpPort				: UINT:=502;		(* (NA) Tcp port *)
	ParamIPAddress				: STRING;           (* (NA) IP address*)
	ParamUnitID					: BYTE;             (* (NA) Unit ID*)
END_VAR

VAR_OUTPUT
	
END_VAR

VAR_INPUT
	
	MesDataExd    	AT %Q*	: UPS_PS10048;

END_VAR


VAR

	FB_ModbusRead	          	: ARRAY[1..4] OF FB_ModbusRead; 
			
	MesBlock1_Temp 				: ARRAY [1..1] OF WORD ; 
	MesBlock2_Temp 				: ARRAY [1..11] OF WORD ; 
	MesBlock3_Temp 				: ARRAY [1..8] OF WORD ; 
	MesBlock4_Temp 				: ARRAY [1..2] OF WORD ; 
	
	AX_ModbusReadAlarm			: ARRAY[1..4] OF BOOL;
	AX_ModbusReadAlarmId		: ARRAY[1..4] OF UDINT;	
END_VAR

